// TwinCAT 3 PLC project Tc3_mxAutomationSample
// ProgramVersion: 3.1.4020.4
// libraries:
//   CmpBitmapPool, * (System)
//   Tc2_Standard, * (Beckhoff Automation GmbH)
//   Tc2_System, * (Beckhoff Automation GmbH)
//   Tc2_Utilities, * (Beckhoff Automation GmbH)
//   Tc3_Module, * (Beckhoff Automation GmbH)
//   Tc3_mxAutomationV3_0, * (Beckhoff Automation GmbH)
//   VisuDialogs, * (System)
// project tree:
//   DUTs/Diagnosis/Enum/ E_ExecMode.TcDUT, E_MoveMode.TcDUT, E_MxAStatus.TcDUT, E_MxA_Error.TcDUT, E_MxA_PCOSError.TcDUT, E_MxA_PLCError.TcDUT, E_MxA_RIError.TcDUT, E_MxA_SIError.TcDUT, E_OriType.TcDUT
//   DUTs/Diagnosis/ ST_AutoExtern.TcDUT, ST_Diag.TcDUT, ST_DiagKRC.TcDUT, ST_ErrorKRC.TcDUT, ST_FromKRC_AutoExtern.TcDUT, ST_FromKRC_P1.TcDUT, ST_GeneralKRCError.TcDUT, ST_ToKRC_AutoExtern.TcDUT, ST_ToKRC_P1.TcDUT, ST_Version.TcDUT
//   DUTs/ Robot_FW.TcDUT, Robot_Position.TcDUT
//   / GlobalTextList.TcGTLO, PlcTask.TcTTO, Visualization Manager.TcVMO (not stored), VISU_TASK.TcTTO
//   GVLs/ GVL_GUI.TcGVL, GVL_PLC.TcGVL, GVL.TcGVL, GVL_SAFETY.TcGVL, GVL_settings.TcGVL
//   POUs/ CheckBounds.TcPOU, Prg_KillHMI.TcPOU (excluded from build)
//   POUs/mxAutomation/ FB_AutoDemo.TcPOU, MAIN.TcPOU, mxA_Motion.TcPOU, Read_Axes_Velocity.TcPOU
//   POUs/Safety/ FB_SafePower.TcPOU, PRG_Safety.TcPOU
//   VISUs/ APP_Settings.TcVIS, diagnostic.TcVIS, communication.TcVIS, ImagePool.TcIPO (not stored), Motion_Axes.TcVIS, Motion_Linear.TcVIS, Motion_FBK.TcVIS, MenuMain.TcVIS, MenuTop.TcVIS, HMI_dmeo.TcVIS, MainScreen.TcVIS
//   VISUs/Text Lists/ CoorSys.TcTLO, GlobalPositions.TcTLO, ToolNumber.TcTLO
// real-time tasks:
//   TASK PlcTask: cycle T#10ms, priority 20, ADS port 350
//   TASK VISU_TASK: cycle T#50000us, priority 30, ADS port 351
// I/O:
//   DEVICE Device 3 (EtherCAT), AmsNetId 5.59.135.8.4.1
//     Box 1 (KRC4 secondary EL6695-1001) [KRC4 secondary EL6695-1001]
//       modules: Module 1 (Sync Inputs), Module 2 (Safety Data Bitf  (8 Byte)), Module 3 (Default IO)
//   DEVICE Device 1 (EtherCAT), AmsNetId 5.59.135.8.2.1
//     Term 2 (EK1200) [EK1200-5000 EtherCAT Power supply (2A E-Bus)]
//       Term 3 (EL1918) [EL1918, 8Ch. Safety Input 24V, TwinSAFE]
//         modules: Module 2 (FSLOGIC)
// variable links:
//   Device 1 (EtherCAT) <-> Device 3 (EtherCAT)/Box 1 (KRC4 secondary EL6695-1001)
//     Term 2 (EK1200)/Term 3 (EL1918)/ConnectionInputs/Message_40 TxPDO <-> Module 2 (Safety Data Bitf  (8 Byte))/Outputs Bitf/FSOE
//   Device 3 (EtherCAT) <-> Device 1 (EtherCAT)/Term 2 (EK1200)/Term 3 (EL1918)
//     Box 1 (KRC4 secondary EL6695-1001)/Module 2 (Safety Data Bitf  (8 Byte))/Inputs Bitf/FSOE <-> ConnectionOutputs/Message_40 RxPDO
//   Tc3_mxAutomationSample Instance <-> Device 1 (EtherCAT)/Term 2 (EK1200)/Term 3 (EL1918)
//     PlcTask Inputs/GVL_SAFETY.ComErr <-> StandardInputs/Standard Out Var 15
//     PlcTask Inputs/GVL_SAFETY.PowerIsOn <-> StandardInputs/Standard Out Var 42
//     PlcTask Outputs/GVL_SAFETY.Ack <-> StandardOutputs/Standard In Var 1
//     PlcTask Outputs/GVL_SAFETY.Restart <-> StandardOutputs/Standard In Var 18
//     PlcTask Outputs/GVL_SAFETY.Run <-> StandardOutputs/Standard In Var 14
//   Tc3_mxAutomationSample Instance <-> Device 3 (EtherCAT)/Box 1 (KRC4 secondary EL6695-1001)
//     PlcTask Inputs/GVL.mxIn <-> Module 3 (Default IO)/Std. In (256 Bytes)/Input DWORD 0
//     PlcTask Inputs/GVL.mxIn @bit {32..2016 step 32} <-> Module 3 (Default IO)/Std. In (256 Bytes)/Input DWORD {1..63}  (63 links)
//     PlcTask Outputs/GVL.mxOut <-> Module 3 (Default IO)/Std. Out (256 Bytes)/Output DWORD 0
//     PlcTask Outputs/GVL.mxOut @bit {32..2016 step 32} <-> Module 3 (Default IO)/Std. Out (256 Bytes)/Output DWORD {1..63}  (63 links)

CONFIGURATION Tc3_mxAutomationSample
    RESOURCE PLC ON TwinCAT3
        TASK PlcTask(INTERVAL := T#10ms, PRIORITY := 20);
        TASK VISU_TASK(INTERVAL := T#50000us, PRIORITY := 30);
        PROGRAM MAIN WITH PlcTask : MAIN;
        PROGRAM VisuElems_Visu_Prg WITH VISU_TASK : VisuElems.Visu_Prg;
    END_RESOURCE
END_CONFIGURATION

// ---- DUTs/Diagnosis/Enum/E_ExecMode.TcDUT
TYPE E_ExecMode :
(
	eEM_Submit 		:= 0, 	//direct execution, 0
	eEM_Aborting	:= 1,	//1
	eEM_Buffered	:= 2	//2
) BYTE;
END_TYPE

// ---- DUTs/Diagnosis/Enum/E_MoveMode.TcDUT
TYPE E_MoveMode :
(
	eMM_MoveAxisAbsolute := 0,
	eMM_MoveRobLinearAbsolute
);
END_TYPE

// ---- DUTs/Diagnosis/Enum/E_MxAStatus.TcDUT
TYPE E_MxAStatus :
(
	eMxA_Invalid := 0,
	eMxA_Error,
	eMxA_ProgramStopped,
	eMxA_StandBy,
	eMxA_Executing,
	eMxA_Aborting
);
END_TYPE

// ---- DUTs/Diagnosis/Enum/E_MxA_Error.TcDUT
TYPE E_MxA_Error :
(
	eMxA_OK 				:= 0, 

	eMxA_SI_InternalError,  	
	eMxA_SI_AssertFailed,		
	eMxA_SI_OvrflwStatRetQueueMain,
	eMxA_SI_OvrflwStatRetQueueTrig,
	eMxA_SI_InvCmdQueueIndex,
	eMxA_SI_InvCmdState,
	eMxA_SI_InvCmdID,
	eMxA_SI_InvMoveType,
	eMxA_SI_TrigFifoFull,
	eMxA_SI_TrigFifoEmpty,
	eMxA_SI_InvTrigFifoIndex,
	eMxA_SI_ExecOfTAfterMiss,
	eMxA_SI_ExecOfTStartMiss,
	eMxA_SI_InvAdvAct,
	eMxA_SI_AbortReq,
	eMxA_SI_TmoutHeartbeatFromPlc 	:= 16,
	eMxA_SI_InvPtpApo 				:= 30,
	eMxA_SI_InvCpApo,
	eMxA_SI_InvBaseNo,
	eMxA_SI_InvToolNo,
	eMxA_SI_InvVelo,
	eMxA_SI_InvAccel,
	eMxA_SI_InvCPtp,
	eMxA_SI_InvCDis,
	eMxA_SI_InvCVelo,
	eMxA_SI_InvCOri,
	eMxA_SI_InvOriType,
	eMxA_SI_PosDataNotInit,
	eMxA_SI_AxisPosDataNotInit,
	eMxA_SI_InvTrigDis,
	eMxA_SI_InvTrigIO,
	eMxA_SI_InvTrigPulse,
	eMxA_SI_InvCircHP,
	eMxA_SI_InvIntIO,
	eMxA_SI_InvIntPrio,
	eMxA_SI_IntNotDecl,
	eMxA_SI_InvIntAct,
	eMxA_SI_InvIONo,
	eMxA_SI_InvPulseDuration,
	eMxA_SI_InvBufferMode,
	eMxA_SI_InvToolNoForDataLoad,
	eMxA_SI_InvAnalogIONo,
	eMxA_SI_InvIpoMode,
	eMxA_SI_InvCircType,
	eMxA_SI_InvFrameData,
	eMxA_SI_InvLodaData,
	eMxA_SI_InvSoftEndRev,
	eMxA_SI_InvIntState,
	eMxA_SI_InvSysVarIndex,
	eMxA_SI_InvSysVarValue,
	eMxA_SI_SysVarNotWritable,
	eMxA_SI_InvRealValue,
	eMxA_SI_ErrorSettingOutput,
	eMxA_SI_ErrorSettingSoftEnd,
	eMxA_SI_InvTechFuncIndex,
	eMxA_SI_InvTechFuncPar,
	eMxA_SI_ParValue,

	eMxA_RI_InternalError		:= 401,	
	eMxA_RI_AssertFailed,
	eMxA_RI_InvCmdID,
	eMxA_RI_InvCmdState,
	eMxA_RI_OvrflwCmdQueue,
	eMxA_RI_IncCmdQueueIndex,
	eMxA_RI_InvCmdPreQueueIndex,
	eMxA_RI_InvWriteQueueIndex,
	eMxA_RI_StatusRetQueueSubmFull,
	eMxA_RI_InvFldbusTelLen,
	eMxA_RI_TmoutAbortReq,
	eMxA_RI_InvChkSumPlcToKrc	:= 412,
	eMxA_RI_InvMoveType,
	eMxA_RI_TmoutHeartbeatFromPlc,	
	eMxA_RI_SysVarNotInit		:= 416,
	eMxA_RI_UndflwOfNibble,
	eMxA_RI_OvrflwOfNibble,
	eMxA_RI_UndflwOfByte,
	eMxA_RI_OvrflwOfByte,
	eMxA_RI_UndflwOfInt16,
	eMxA_RI_OvrflwOfInt16,
	eMxA_RI_UndflwOfInt32,
	eMxA_RI_OvrflwOfInt32,
	eMxA_RI_UndflwOfReal,
	eMxA_RI_OvrflwOfReal,
	eMxA_RI_InvPtpApo 			:= 430,
	eMxA_RI_InvCpApo,
	eMxA_RI_InvBasNo,
	eMxA_RI_InvToolNo,
	eMxA_RI_InvVelo,
	eMxA_RI_InvAccel,
	eMxA_RI_InvCPtp,
	eMxA_RI_InvCDis,
	eMxA_RI_InvCVelo,
	eMxA_RI_InvCOri,
	eMxA_RI_InvOriType,
	eMxA_RI_PosDataNotInit,
	eMxA_RI_AxisPosDataNotInit,
	eMxA_RI_InvTrigDis,
	eMxA_RI_InvTrigIO,
	eMxA_RI_InvTrigPulse,
	eMxA_RI_InvCircHP,
	eMxA_RI_InvIntIO,
	eMxA_RI_InvIntPrio,
	eMxA_RI_IntNotDecl,
	eMxA_RI_InvIntAct,
	eMxA_RI_InvIONo,
	eMxA_RI_InvPulseDuration,
	eMxA_RI_InvBufferMode,
	eMxA_RI_InvToolNoForDataLoad,
	eMxA_RI_InvAnalogIONo,
	eMxA_RI_InvIpoMode,
	eMxA_RI_InvCircType,
	eMxA_RI_InvFrameData,
	eMxA_RI_InvLodaData,
	eMxA_RI_InvSoftEndRev,
	eMxA_RI_InvIntState,
	eMxA_RI_InvSysVarIndex,
	eMxA_RI_InvSysVarValue,
	eMxA_RI_SysVarNotWritable,
	eMxA_RI_InvRealValue,
	eMxA_RI_ErrorSettingOutput,
	eMxA_RI_ErrorSettingSoftEnd,
	eMxA_RI_InvTechFuncIndex,
	eMxA_RI_InvTechFuncPar,
	eMxA_RI_ParValue,

	eMxA_PLC_InternalError		:= 501,
	eMxA_PLC_InvBufferMode,
	eMxA_PLC_InvMxaVer,
	eMxA_PLC_InvOverride,
	eMxA_PLC_InvGrpRefIndexReached,
	eMxA_PLC_InvGrpPrefIndex,
	eMxA_PLC_InvFBOrder,
	eMxA_PLC_ConnectNotInit,
	eMxA_PLC_NoConnectToKrc,
	eMxA_PLC_TmoutHeartbeatFromKrc,
	eMxA_PLC_TmoutCmdItfBlocked,
	eMxA_PLC_InvChkSumKrcToPlc,
	eMxA_PLC_InvPosIndex,
	eMxA_PLC_PosActInv,
	eMxA_PLC_PNetError,
	eMxA_PLC_ENetIpError,
	eMxA_PLC_InvCmdSize,
	
	eMxA_PCOS_InternalError		:= 701,
	eMxA_PCOS_AssertFailed,
	eMxA_PCOS_InvCmdID,
	eMxA_PCOS_InvHeaderData,
	eMxA_PCOS_InvChkSumPlcToKrc	:= 712,
	eMxA_PCOS_InvMoveType,
	eMxA_PCOS_InvPtpApo			:= 730,
	eMxA_PCOS_InvCpApo,
	eMxA_PCOS_InvBasNo,
	eMxA_PCOS_InvToolNo,
	eMxA_PCOS_InvVelo,
	eMxA_PCOS_InvAccel,
	eMxA_PCOS_InvCPtp,
	eMxA_PCOS_InvCDis,
	eMxA_PCOS_InvCVelo,
	eMxA_PCOS_InvCOri,
	eMxA_PCOS_InvOriType,
	eMxA_PCOS_PosDataNotInit,
	eMxA_PCOS_AxisPosDataNotInit,
	eMxA_PCOS_InvTrigDis,
	eMxA_PCOS_InvTrigIO,
	eMxA_PCOS_InvTrigPulse,
	eMxA_PCOS_InvCircHP,
	eMxA_PCOS_InvIntIO,
	eMxA_PCOS_InvIntPrio,
	eMxA_PCOS_InvIntAct		:= 750,
	eMxA_PCOS_InvIONo,
	eMxA_PCOS_InvPulseDuration,
	eMxA_PCOS_InvBufferMode,
	eMxA_PCOS_InvToolNoForDataLoad,
	eMxA_PCOS_InvAnalogIONo,
	eMxA_PCOS_InvIpoMode,
	eMxA_PCOS_InvCircType,
	eMxA_PCOS_InvFrameData,
	eMxA_PCOS_InvLodaData,
	eMxA_PCOS_InvSoftEndRev,
	eMxA_PCOS_InvRealValue	:= 765,
	eMxA_PCOS_ParValue		:= 770
) DINT;
END_TYPE

// ---- DUTs/Diagnosis/Enum/E_MxA_PCOSError.TcDUT
TYPE E_MxA_PCOSError :
(
	eMxA_OK 				:= 0, 	
	eMxA_InternalError		:= 701,
	eMxA_AssertFailed,
	eMxA_InvCmdID,
	eMxA_InvHeaderData,
	eMxA_InvChkSumPlcToKrc	:= 712,
	eMxA_InvMoveType,
	eMxA_InvPtpApo			:= 730,
	eMxA_InvCpApo,
	eMxA_InvBasNo,
	eMxA_InvToolNo,
	eMxA_InvVelo,
	eMxA_InvAccel,
	eMxA_InvCPtp,
	eMxA_InvCDis,
	eMxA_InvCVelo,
	eMxA_InvCOri,
	eMxA_InvOriType,
	eMxA_PosDataNotInit,
	eMxA_AxisPosDataNotInit,
	eMxA_InvTrigDis,
	eMxA_InvTrigIO,
	eMxA_InvTrigPulse,
	eMxA_InvCircHP,
	eMxA_InvIntIO,
	eMxA_InvIntPrio,
	eMxA_InvIntAct		:= 750,
	eMxA_InvIONo,
	eMxA_InvPulseDuration,
	eMxA_InvBufferMode,
	eMxA_InvToolNoForDataLoad,
	eMxA_InvAnalogIONo,
	eMxA_InvIpoMode,
	eMxA_InvCircType,
	eMxA_InvFrameData,
	eMxA_InvLodaData,
	eMxA_InvSoftEndRev,
	eMxA_InvRealValue	:= 765,
	eMxA_ParValue		:= 770
) DINT;
END_TYPE

// ---- DUTs/Diagnosis/Enum/E_MxA_PLCError.TcDUT
TYPE E_MxA_PLCError :
(
	eMxA_OK 				:= 0, 	
	eMxA_InternalError		:= 501,
	eMxA_InvBufferMode,
	eMxA_InvMxaVer,
	eMxA_InvOverride,
	eMxA_InvGrpRefIndexReached,
	eMxA_InvGrpPrefIndex,
	eMxA_InvFBOrder,
	eMxA_ConnectNotInit,
	eMxA_NoConnectToKrc,
	eMxA_TmoutHeartbeatFromKrc,
	eMxA_TmoutCmdItfBlocked,
	eMxA_InvChkSumKrcToPlc,
	eMxA_InvPosIndex,
	eMxA_PosActInv,
	eMxA_PNetError,
	eMxA_ENetIpError,
	eMxA_InvCmdSize
) DINT;
END_TYPE

// ---- DUTs/Diagnosis/Enum/E_MxA_RIError.TcDUT
TYPE E_MxA_RIError :
(
	eMxA_OK 				:= 0, 	
	eMxA_InternalError		:= 401,	
	eMxA_AssertFailed,
	eMxA_InvCmdID,
	eMxA_InvCmdState,
	eMxA_OvrflwCmdQueue,
	eMxA_IncCmdQueueIndex,
	eMxA_InvCmdPreQueueIndex,
	eMxA_InvWriteQueueIndex,
	eMxA_StatusRetQueueSubmFull,
	eMxA_InvFldbusTelLen,
	eMxA_TmoutAbortReq,
	eMxA_InvChkSumPlcToKrc	:= 412,
	eMxA_InvMoveType,
	eMxA_TmoutHeartbeatFromPlc,	
	eMxA_SysVarNotInit		:= 416,
	eMxA_UndflwOfNibble,
	eMxA_OvrflwOfNibble,
	eMxA_UndflwOfByte,
	eMxA_OvrflwOfByte,
	eMxA_UndflwOfInt16,
	eMxA_OvrflwOfInt16,
	eMxA_UndflwOfInt32,
	eMxA_OvrflwOfInt32,
	eMxA_UndflwOfReal,
	eMxA_OvrflwOfReal,
	eMxA_InvPtpApo 			:= 430,
	eMxA_InvCpApo,
	eMxA_InvBasNo,
	eMxA_InvToolNo,
	eMxA_InvVelo,
	eMxA_InvAccel,
	eMxA_InvCPtp,
	eMxA_InvCDis,
	eMxA_InvCVelo,
	eMxA_InvCOri,
	eMxA_InvOriType,
	eMxA_PosDataNotInit,
	eMxA_AxisPosDataNotInit,
	eMxA_InvTrigDis,
	eMxA_InvTrigIO,
	eMxA_InvTrigPulse,
	eMxA_InvCircHP,
	eMxA_InvIntIO,
	eMxA_InvIntPrio,
	eMxA_IntNotDecl,
	eMxA_InvIntAct,
	eMxA_InvIONo,
	eMxA_InvPulseDuration,
	eMxA_InvBufferMode,
	eMxA_InvToolNoForDataLoad,
	eMxA_InvAnalogIONo,
	eMxA_InvIpoMode,
	eMxA_InvCircType,
	eMxA_InvFrameData,
	eMxA_InvLodaData,
	eMxA_InvSoftEndRev,
	eMxA_InvIntState,
	eMxA_InvSysVarIndex,
	eMxA_InvSysVarValue,
	eMxA_SysVarNotWritable,
	eMxA_InvRealValue,
	eMxA_ErrorSettingOutput,
	eMxA_ErrorSettingSoftEnd,
	eMxA_InvTechFuncIndex,
	eMxA_InvTechFuncPar,
	eMxA_ParValue
) DINT;
END_TYPE

// ---- DUTs/Diagnosis/Enum/E_MxA_SIError.TcDUT
TYPE E_MxA_SIError :
(
	eMxA_OK 					:= 0, 	
	eMxA_InternalError,  	
	eMxA_AssertFailed,		
	eMxA_OvrflwStatRetQueueMain,
	eMxA_OvrflwStatRetQueueTrig,
	eMxA_InvCmdQueueIndex,
	eMxA_InvCmdState,
	eMxA_InvCmdID,
	eMxA_InvMoveType,
	eMxA_TrigFifoFull,
	eMxA_TrigFifoEmpty,
	eMxA_InvTrigFifoIndex,
	eMxA_ExecOfTAfterMiss,
	eMxA_ExecOfTStartMiss,
	eMxA_InvAdvAct,
	eMxA_AbortReq,
	eMxA_TmoutHeartbeatFromPlc 	:= 16,
	eMxA_InvPtpApo 				:= 30,
	eMxA_InvCpApo,
	eMxA_InvBaseNo,
	eMxA_InvToolNo,
	eMxA_InvVelo,
	eMxA_InvAccel,
	eMxA_InvCPtp,
	eMxA_InvCDis,
	eMxA_InvCVelo,
	eMxA_InvCOri,
	eMxA_InvOriType,
	eMxA_PosDataNotInit,
	eMxA_AxisPosDataNotInit,
	eMxA_InvTrigDis,
	eMxA_InvTrigIO,
	eMxA_InvTrigPulse,
	eMxA_InvCircHP,
	eMxA_InvIntIO,
	eMxA_InvIntPrio,
	eMxA_IntNotDecl,
	eMxA_InvIntAct,
	eMxA_InvIONo,
	eMxA_InvPulseDuration,
	eMxA_InvBufferMode,
	eMxA_InvToolNoForDataLoad,
	eMxA_InvAnalogIONo,
	eMxA_InvIpoMode,
	eMxA_InvCircType,
	eMxA_InvFrameData,
	eMxA_InvLodaData,
	eMxA_InvSoftEndRev,
	eMxA_InvIntState,
	eMxA_InvSysVarIndex,
	eMxA_InvSysVarValue,
	eMxA_SysVarNotWritable,
	eMxA_InvRealValue,
	eMxA_ErrorSettingOutput,
	eMxA_ErrorSettingSoftEnd,
	eMxA_InvTechFuncIndex,
	eMxA_InvTechFuncPar,
	eMxA_ParValue
) DINT;
END_TYPE

// ---- DUTs/Diagnosis/Enum/E_OriType.TcDUT
TYPE E_OriType :
(
	eOT_Var := 0,
	eOT_Constant,
	eOT_Joint
);
END_TYPE

// ---- DUTs/Diagnosis/ST_AutoExtern.TcDUT
TYPE ST_AutoExtern :
STRUCT
	bValid				: bool;
	bRcReady			: BOOL;
	bAlarmStop			: BOOL;
	bUserSAFE			: BOOL;
	bPeriReady			: BOOL;
	bRobCal				: BOOL;
	bIoActConf			: BOOL;
	bStopMess			: BOOL;
	bIntEStop			: BOOL;
	bProAct				: BOOL;
	bApplRun			: BOOL;
	bProMove			: BOOL;
	bOnPath				: BOOL;
	bNearPosRet			: BOOL;
	bRobStopped			: BOOL;
	bT1					: BOOL;
	bT2					: BOOL;
	bAUT				: BOOL;
	bEXT				: BOOL;
END_STRUCT
END_TYPE

// ---- DUTs/Diagnosis/ST_Diag.TcDUT
TYPE ST_Diag :
STRUCT
	//KRC diag
	stDiagKRC			: ST_DiagKRC;	
	bDiagKRCError       : BOOL;
	nDiagKRCErrorID     : E_MxA_Error;
		
	//MXA error
	bMXAError           : BOOL;
	nMXAErrorID         : E_MxA_Error;
	
	//MXA status
	nMXAStatus       	: E_MxAStatus;
	bMXAStatusError     : BOOL;
	nMXAStatusErrorID   : E_MxA_Error;

	//KRC error
	stErrorKRC			: ST_ErrorKRC;
	bErrorKRCDone       : BOOL;
	bErrorKRCError      : BOOL;
	nErrorKRCErrorID    : E_MxA_Error;
END_STRUCT
END_TYPE

// ---- DUTs/Diagnosis/ST_DiagKRC.TcDUT
TYPE ST_DiagKRC :
STRUCT
	bValid         		: BOOL;
	nQueueCount         : INT;
	bPosActValid        : BOOL;
	bBrakeActive        : BOOL;
	nSubmitHeartbeat    : INT;
	nSubmitCyc_Act      : INT;
	nSubmitCyc_Min      : INT;
	nSubmitCyc_Max      : INT;
	nSubmitCyc_Avg      : INT;
	nActivePosOrderID   : DINT;
	nActiveOrderIDB     : DINT;
	nAvg_Duration       : DINT; 
	nPCOSHeartbeat 	 	: INT;   
	nPCOSCyc_Act   	 	: INT;
	nPCOSCyc_Min    	: INT;
	nPCOSCyc_Max  	  	: INT;
	nPCOSCyc_Avg    	: INT;
	nErrorID_RI         : E_MxA_RIError;
	nErrorID_SI         : E_MxA_RIError;
	nErrorID_PLC        : E_MxA_PLCError;
	nErrorID_PCOS       : E_MxA_PCOSError;
END_STRUCT
END_TYPE

// ---- DUTs/Diagnosis/ST_ErrorKRC.TcDUT
TYPE ST_ErrorKRC :
STRUCT
	bStopMessage   		: BOOL;
	nMessageCount 		: INT;
	nMessage     		: ARRAY [1..10] OF E_MxA_Error;
END_STRUCT
END_TYPE

// ---- DUTs/Diagnosis/ST_FromKRC_AutoExtern.TcDUT
TYPE ST_FromKRC_AutoExtern :
STRUCT
	bRcReady			: BOOL;	//0.0
	bAlarmStop			: BOOL;	//0.1
	bUserSAFE			: BOOL;	//0.2
	bPeriReady			: BOOL;	//0.3
	bRobCal				: BOOL;	//0.4
	bIoActConf			: BOOL;	//0.5
	bStopMess			: BOOL;	//0.6
	bPgNoFBitRefl		: BOOL;	//0.7
	
	bIntEStop			: BOOL;	//1.0
	bProAct				: BOOL;	//1.1
	bPgNoReq			: BOOL;	//1.2
	bApplRun			: BOOL;	//1.3
	bProMove			: BOOL;	//1.4
	bInHome				: BOOL;	//1.5
	bOnPath				: BOOL;	//1.6
	bNearPosRet			: BOOL;	//1.7
	
	bRobStopped			: BOOL;	//2.0
	bT1					: BOOL;	//2.1
	bT2					: BOOL;	//2.2
	bAUT				: BOOL;	//2.3
	bEXT				: BOOL;	//2.4
	bBrakeTestMonTime	: BOOL;	//2.5
	bBrakeTestReqInt	: BOOL;	//2.6
	bBrakeTestWork		: BOOL;	//2.7
	
	bBrakeTestOK		: BOOL;	//3.0
	bBrakeTestWarn		: BOOL;	//3.1
	bReserve2075		: BOOL;	//3.2
	bBrakeActive		: BOOL;	//3.3
	bKcpConnect			: BOOL;	//3.4
	bTouchUp			: BOOL;	//3.5
	bMasTestReqInt		: BOOL;	//3.6
	bMasTestSwitchOK	: BOOL;	//3.7
END_STRUCT
END_TYPE

// ---- DUTs/Diagnosis/ST_FromKRC_P1.TcDUT
{attribute 'pack_mode' := '1'}
TYPE ST_FromKRC_P1 :
STRUCT
	nStatusDw 			: DWORD;	//0
	nHeartbeatSubmit 	: BYTE;		//4		heartbeat from KRC 1..245
	nInVal_1_8			: BYTE;		//5		Actual Value of Inputs $IN[1]..$IN[8]
	nTouchUpPosNo		: INT;		//6		Position Number for TouchUp (UserTech)
	nSR_Order1_ID		: DINT;		//8		Order ID for feedback of status information
	nSR_Order2_ID		: DINT;		//12	Order ID for feedback of status information
	nSR_Order3_ID		: DINT;		//16	Order ID for feedback of status information
	nSR_Order4_ID		: DINT;		//20	Order ID for feedback of status information
	nSR_Order5_ID		: DINT;		//24	Order ID for feedback of status information
	nSR_Order6_ID		: DINT;		//28	Order ID for feedback of status information
	nSR_Order7_ID		: DINT;		//32	Order ID for feedback of status information
	nSR_Order8_ID		: DINT;		//36	Order ID for feedback of status information
	nSR_Order9_ID		: DINT;		//40	Order ID for feedback of status information
	nSR_Order10_ID		: DINT;		//44	Order ID for feedback of status information
	nSR_Order1_State	: BYTE;		//48	status feedback (in combination with nSR_Order1_ID)	
	nSR_Order2_State	: BYTE;		//49	status feedback (in combination with nSR_Order2_ID)	
	nSR_Order3_State	: BYTE;		//50	status feedback (in combination with nSR_Order3_ID)	
	nSR_Order4_State	: BYTE;		//51	status feedback (in combination with nSR_Order4_ID)	
	nSR_Order5_State	: BYTE;		//52	status feedback (in combination with nSR_Order5_ID)	
	nSR_Order6_State	: BYTE;		//53	status feedback (in combination with nSR_Order6_ID)	
	nSR_Order7_State	: BYTE;		//54	status feedback (in combination with nSR_Order7_ID)	
	nSR_Order8_State	: BYTE;		//55	status feedback (in combination with nSR_Order8_ID)	
	nSR_Order9_State	: BYTE;		//56	status feedback (in combination with nSR_Order9_ID)	
	nSR_Order10_State	: BYTE;		//57	status feedback (in combination with nSR_Order10_ID)	
	bPosActValid		: BOOL;		//58.0	Position data valid (SAK)
	nHeartbeatPCOS		: BYTE;		//59	heartbeat from PCOS 1..245
	nOverride			: BYTE;		//60	SysVar $OV_PRO
	fPosActX			: REAL;		//61	SysVar $POS_ACT.X
	fPosActY			: REAL;		//65	SysVar $POS_ACT.Y
	fPosActZ			: REAL;		//69	SysVar $POS_ACT.Z
	fPosActA			: REAL;		//73	SysVar $POS_ACT.A
	fPosActB			: REAL;		//77	SysVar $POS_ACT.B
	fPosActC			: REAL;		//81	SysVar $POS_ACT.C
	nPosActStatus		: DINT;		//85	SysVar $POS_ACT.S
	nPosActTurns		: BYTE;		//89	SysVar $POS_ACT.T
	nToolAct			: SINT;		//90	SysVar $ACT_TOOL_C
	nBaseAct			: SINT;		//91	SysVar $ACT_BASE_C
	nIpoMode			: BYTE;		//92	SysVar $IPO_MODE_C
	fAxisAct_A1			: REAL;		//93	SysVar $AXIS_ACT.A1
	fAxisAct_A2			: REAL;		//97	SysVar $AXIS_ACT.A2
	fAxisAct_A3			: REAL;		//101	SysVar $AXIS_ACT.A3
	fAxisAct_A4			: REAL;		//105	SysVar $AXIS_ACT.A4
	fAxisAct_A5			: REAL;		//109	SysVar $AXIS_ACT.A5
	fAxisAct_A6			: REAL;		//113	SysVar $AXIS_ACT.A6
	fAxisAct_A7			: REAL;		//117	SysVar $AXIS_ACT.A7
	fAxisAct_A8			: REAL;		//121	SysVar $AXIS_ACT.A8
	fAxisAct_A9			: REAL;		//125	SysVar $AXIS_ACT.A9
	fAxisAct_A10		: REAL;		//129	SysVar $AXIS_ACT.A10
	fAxisAct_A11		: REAL;		//133	SysVar $AXIS_ACT.A11
	fAxisAct_A12		: REAL;		//137	SysVar $AXIS_ACT.A12
	fVelAct				: REAL;		//141	SysVar $VEL_ACT
	nVelAxis_A1			: SINT;		//145	SysVar $VEL_AXIS_ACT[1]
	nVelAxis_A2			: SINT;		//146	SysVar $VEL_AXIS_ACT[2]
	nVelAxis_A3			: SINT;		//147	SysVar $VEL_AXIS_ACT[3]
	nVelAxis_A4			: SINT;		//148	SysVar $VEL_AXIS_ACT[4]
	nVelAxis_A5			: SINT;		//149	SysVar $VEL_AXIS_ACT[5]
	nVelAxis_A6			: SINT;		//150	SysVar $VEL_AXIS_ACT[6]
	nVelAxis_A7			: SINT;		//151	SysVar $VEL_AXIS_ACT[7]
	nVelAxis_A8			: SINT;		//152	SysVar $VEL_AXIS_ACT[8]
	nVelAxis_A9			: SINT;		//153	SysVar $VEL_AXIS_ACT[9]
	nVelAxis_A10		: SINT;		//154	SysVar $VEL_AXIS_ACT[10]
	nVelAxis_A11		: SINT;		//155	SysVar $VEL_AXIS_ACT[11]
	nVelAxis_A12		: SINT;		//156	SysVar $VEL_AXIS_ACT[12]
	nGroupState			: BYTE;		//157	see state diagram
	nErrorId			: INT;		//158	error id from main loop or interrupt
	nErrorSubId			: INT;		//160	error id from submit interpreter
	nActivePosOrderId	: DINT;		//162	order id of active move cmd
	nActiveOrderIdB		: DINT;		//166	active order id in preparation
	nQueueCount			: BYTE;		//170	current amount of functions in buffer
	nIR_Status_1_2		: BYTE;		//171	status of interrupt 1 and 2
	nIR_Status_3_4		: BYTE;		//172	status of interrupt 3 and 4
	nIR_Status_5_6		: BYTE;		//173	status of interrupt 5 and 6
	nIR_Status_7_8		: BYTE;		//174	status of interrupt 7 and 8
	nErrorIdPCOS		: BYTE;		//175	error id of ProConOS
	nFreeForMove		: BYTE;		//176	reserved for ProConOS
	nTransmissionNoNet	: BYTE;		//177	acknowledge of transmission number
	nOrderIdRet			: DINT;		//178	acknowledge take data of cmd
	nCmdIdRet			: DINT;		//182	acknowledge take data of cmd
	nCmdDataRetCS		: DINT;		//186	checksum data feedback
	nReserved190		: DINT;		//190	reserved
	fCmdDataRet1		: REAL;		//194	command dependent	
	fCmdDataRet2		: REAL;		//198	command dependent	
	fCmdDataRet3		: REAL;		//202	command dependent	
	fCmdDataRet4		: REAL;		//206	command dependent	
	fCmdDataRet5		: REAL;		//210	command dependent	
	fCmdDataRet6		: REAL;		//214	command dependent	
	fCmdDataRet7		: REAL;		//218	command dependent	
	fCmdDataRet8		: REAL;		//222	command dependent	
	fCmdDataRet9		: REAL;		//226	command dependent	
	fCmdDataRet10		: REAL;		//230	command dependent	
	fCmdDataRet11		: REAL;		//234	command dependent	
	fCmdDataRet12		: REAL;		//238	command dependent
	nReserve242			: DINT;		//242	reserved	
	nReserve246			: ARRAY [1..10] OF BYTE; //246..255
END_STRUCT
END_TYPE

// ---- DUTs/Diagnosis/ST_GeneralKRCError.TcDUT
TYPE ST_GeneralKRCError :
STRUCT
	nErrorId 			: DINT;
	bNoHeartbeatKrc 	: BOOL;
	bNoHeartbeatPCOS 	: BOOL;
	bNotOnline 			: BOOL;
	bNotInitialized 	: BOOL;
	bNoOpModeExt 		: BOOL;
	bNoMoveEnable		: BOOL;
	bUserSafeNotOK		: BOOL;
	bKrcErrorActive 	: BOOL;
	bDrivesNotReady		: BOOL; 
	bNoProgActive		: BOOL;
END_STRUCT
END_TYPE

// ---- DUTs/Diagnosis/ST_ToKRC_AutoExtern.TcDUT
TYPE ST_ToKRC_AutoExtern :
STRUCT
	bPgNo_FBit			: BOOL;	//0.0
	bPgNo_Bit1			: BOOL;	//0.1
	bPgNo_Bit2			: BOOL;	//0.2
	bPgNo_Bit3			: BOOL;	//0.3
	bPgNo_Bit4			: BOOL;	//0.4
	bPgNo_Bit5			: BOOL;	//0.5
	bPgNo_Bit6			: BOOL;	//0.6
	bPgNo_Bit7			: BOOL;	//0.7
	
	bPgNo_Parity		: BOOL;	//1.0
	bPgNo_Valid			: BOOL;	//1.1
	bExtStart			: BOOL;	//1.2
	bMoveEnable			: BOOL;	//1.3
	bConfMess			: BOOL;	//1.4
	bDrivesOff			: BOOL;	//1.5
	bDrivesOn			: BOOL;	//1.6
	bMasteringTestReqExt: BOOL;	//1.7
	
	bBrakeTestReqExt	: BOOL;	//2.0
	bReserve_2_1_3_7	: ARRAY[1..15] OF BOOL; //2.1 - 3.7
	
	bReset				: BOOL;	//4.0	choose cell program with rising edge
	bBrake				: BOOL;	//4.1	brake command (KRC interrupt)
	bBrakeF				: BOOL;	//4.2	brakeF command (KRC interrupt)
	bReleaseBrake		: BOOL;	//4.3	release brake after brake command
	bShowTrace			: BOOL;	//4.4	show diag messages in message window
	bMessageReset		: BOOL;	//4.5	message aknowledge of error messages of mxAutomation package
	bReserve_4_6		: BOOL;	//4.6
	bWriteOut_1to8		: BOOL;	//4.7	write request for outputs 1 to 8
	
	bOutVal1			: BOOL;	//5.0	setvalue for $OUT[1]
	bOutVal2			: BOOL;	//5.1	setvalue for $OUT[2]
	bOutVal3			: BOOL;	//5.2	setvalue for $OUT[3]
	bOutVal4			: BOOL;	//5.3	setvalue for $OUT[4]
	bOutVal5			: BOOL;	//5.4	setvalue for $OUT[5]
	bOutVal6			: BOOL;	//5.5	setvalue for $OUT[6]
	bOutVal7			: BOOL;	//5.6	setvalue for $OUT[7]
	bOutVal8			: BOOL;	//5.7	setvalue for $OUT[8]
	
	bReserve_6_0_7_7	: ARRAY[1..16] OF BOOL; //6.0 - 7.7
END_STRUCT
END_TYPE

// ---- DUTs/Diagnosis/ST_ToKRC_P1.TcDUT
{attribute 'pack_mode' := '1'}
TYPE ST_ToKRC_P1 :
STRUCT
	nControlLw			: LWORD;	//0
	nHeartbeat			: BYTE;		//8		heartbeat KRC and ProConOS, 1..254
	nOverride			: BYTE;		//9		override of extern
	nPlcVersionMajor	: BYTE;		//10	major PLC version
	nPlcVersionMinor	: BYTE;		//11	minor PLC version
	nSR_Order1_IdRet	: DINT;		//12	order id for acknowledge of status feedback
	nSR_Order2_IdRet	: DINT;		//16	order id for acknowledge of status feedback
	nSR_Order3_IdRet	: DINT;		//20	order id for acknowledge of status feedback
	nSR_Order4_IdRet	: DINT;		//24	order id for acknowledge of status feedback
	nSR_Order5_IdRet	: DINT;		//28	order id for acknowledge of status feedback
	nSR_Order6_IdRet	: DINT;		//32	order id for acknowledge of status feedback
	nSR_Order7_IdRet	: DINT;		//36	order id for acknowledge of status feedback
	nSR_Order8_IdRet	: DINT;		//40	order id for acknowledge of status feedback
	nSR_Order9_IdRet	: DINT;		//44	order id for acknowledge of status feedback
	nSR_Order10_IdRet	: DINT;		//48	order id for acknowledge of status feedback
	nSR_Order1_State	: BYTE;		//52	order id for acknowledge of status feedback
	nSR_Order2_State	: BYTE;		//53	order id for acknowledge of status feedback
	nSR_Order3_State	: BYTE;		//54	order id for acknowledge of status feedback
	nSR_Order4_State	: BYTE;		//55	order id for acknowledge of status feedback
	nSR_Order5_State	: BYTE;		//56	order id for acknowledge of status feedback
	nSR_Order6_State	: BYTE;		//57	order id for acknowledge of status feedback
	nSR_Order7_State	: BYTE;		//58	order id for acknowledge of status feedback
	nSR_Order8_State	: BYTE;		//59	order id for acknowledge of status feedback
	nSR_Order9_State	: BYTE;		//60	order id for acknowledge of status feedback
	nSR_Order10_State	: BYTE;		//61	order id for acknowledge of status feedback
	nTransmissionNO1	: BYTE;		//62	1..254: transmission number, 0: no active transmission
	nTransmissionType	: BYTE;		//63	1: Part 1/1, 2: Part 1/2, 3: Part 2/2, 4: Part 1/3, 5: Part 2/3, 6: Part 3/3
	nOrderId			: DINT;		//64	unique order id, incr. with rising edge on bExecute on FB, 1..2^31-1
	nCmdId				: BYTE;		//68	command id
	eExecMode			: E_ExecMode;//69	Enum Byte: 0: Submit (direct execution in submit), 1: aborting, 2: buffered
	nCheckSum			: DWORD;	//70	XOR checksum of command data
	nBoolValues1		: WORD;		//74	bool parameter values 1-15, 16-30, 31-45
	nCmdParInt1			: DINT;		//76	integer parameter 1, 16, 31
	nCmdParInt2			: DINT;		//80	integer parameter 2, 17, 32
	nCmdParInt3			: DINT;		//84	integer parameter 3, 18, 33
	nCmdParInt4			: DINT;		//88	integer parameter 4, 19, 34
	nCmdParInt5			: DINT;		//92	integer parameter 5, 20, 35
	nCmdParInt6			: DINT;		//96	integer parameter 6, 21, 36
	nCmdParInt7			: DINT;		//100	integer parameter 7, 22, 37
	nCmdParInt8			: DINT;		//104	integer parameter 8, 23, 38
	nCmdParInt9			: DINT;		//108	integer parameter 9, 24, 39
	nCmdParInt10		: DINT;		//112	integer parameter 10, 25, 40
	nCmdParInt11		: DINT;		//116	integer parameter 11, 26, 41
	nCmdParInt12		: DINT;		//120	integer parameter 12, 27, 42
	nCmdParInt13		: DINT;		//124	integer parameter 13, 28, 43
	nCmdParInt14		: DINT;		//128	integer parameter 14, 29, 44
	nCmdParInt15		: DINT;		//132	integer parameter 15, 30, 45
	fCmdParReal1		: REAL;		//136	real parameter 1, 16, 31
	fCmdParReal2		: REAL;		//140	real parameter 2, 17, 32
	fCmdParReal3		: REAL;		//144	real parameter 3, 18, 33
	fCmdParReal4		: REAL;		//148	real parameter 4, 19, 34
	fCmdParReal5		: REAL;		//152	real parameter 5, 20, 35
	fCmdParReal6		: REAL;		//156	real parameter 6, 21, 36
	fCmdParReal7		: REAL;		//160	real parameter 7, 22, 37
	fCmdParReal8		: REAL;		//164	real parameter 8, 23, 38
	fCmdParReal9		: REAL;		//168	real parameter 9, 24, 39
	fCmdParReal10		: REAL;		//172	real parameter 10, 25, 40
	fCmdParReal11		: REAL;		//176	real parameter 11, 26, 41
	fCmdParReal12		: REAL;		//180	real parameter 12, 27, 42
	fCmdParReal13		: REAL;		//184	real parameter 13, 28, 43
	fCmdParReal14		: REAL;		//188	real parameter 14, 29, 44
	fCmdParReal15		: REAL;		//192	real parameter 15, 30, 45
	nTransmissionNO2	: BYTE;		//196	transmission number for consistency check, need to match with nTransmissionNO1
	nReserved197		: ARRAY [1..59] OF BYTE;	
END_STRUCT
END_TYPE

// ---- DUTs/Diagnosis/ST_Version.TcDUT
TYPE ST_Version :
STRUCT
	nMajor    		: DINT;
	nMinor    		: DINT;
	nBuild 			: DINT;
	nRevision 		: DINT;
	sVersion		: STRING;
END_STRUCT
END_TYPE

// ---- DUTs/Robot_FW.TcDUT
TYPE Robot_FW :
	
STRUCT
	FW_Version :DINT;
	FW_Major:DINT;
	FW_Minor:DINT;
	
END_STRUCT


END_TYPE

// ---- DUTs/Robot_Position.TcDUT
TYPE Robot_Position :
	

STRUCT
	
p1:REAL;
p2:REAL;
p3:REAL;
p4:REAL;
p5:REAL;
p6:REAL;

END_STRUCT


END_TYPE

// ---- GVLs/GVL_GUI.TcGVL
{attribute 'qualified_only'}
VAR_GLOBAL
	
	LinearTargetCommand :STRING;
	GlobalPositionString :STRING;

	
END_VAR

// ---- GVLs/GVL_PLC.TcGVL
{attribute 'qualified_only'}
VAR_GLOBAL
	
	Int_windowsCounter: ULINT;
	Str_windowsCounter: STRING;
	
	
	ReadWindowsTime : fb_localsystemTime;
	String_WindowsTime: STRING;
	Time_SystemTime : TIMESTRUCT;
	
END_VAR

// ---- GVLs/GVL.TcGVL
{attribute 'qualified_only'}
VAR_GLOBAL
	
//=====================================
// mxAutomation
//=====================================	

	mxIn					AT%I* 	: ARRAY[0..63] OF DWORD;
	mxOut 					AT%Q* 	: ARRAY[0..63] OF DWORD;
	
	nAxisIndex						: INT := 1;  // Robot number one, may be any unique number between 1..5
	nOverrideGlobal					: INT;
	
	stCoordSys						: COORDSYS;
	stApprox						: APO;
	
	HMI_ActualCartPos				: E6POS;
	HMI_ActualAxisPosition			: E6AXIS;
	
	HMI_AutoStart					: BOOL;
	HMI_MessageReset				: BOOL;
	
	HMI_AutoEXT						: BOOL;
	HMI_DrivesNotReady				: BOOL;
	
	HMI_Error_ProConOS				: BOOL;
	HMI_Error_SINT					: BOOL;
	HMI_Error_General				: BOOL;
	HMI_Error_General_ID			: DINT;
	
	HMI_WriteLoadData				: BOOL;
	HMI_LOAD						: INT;
	HMI_TOOL						: INT;
	HMI_BASE						: INT;
	
	HMI_TouchUpStoreNow				: BOOL;
	HMI_TouchUpIndex				: INT;
	
	in_MOVE_ENABLE					: BOOL;
	in_CONF_MESS					: BOOL;
	in_DRIVES_ON					: BOOL;
	in_DRIVES_OFF					: BOOL;
	in_EXT_START					: BOOL;
	in_ENABLE_T1					: BOOL;
	in_ENABLE_T2					: BOOL;
	in_ENABLE_AUT					: BOOL;
	in_ENABLE_EXT					: BOOL;
	
	out_ALARM_STOP					: BOOL;
	out_USER_SAFE					: BOOL;
	
	
END_VAR 
VAR_GLOBAL RETAIN
	aPosArray	 					: POSITION_ARRAY;
	LinearArray 					: POSITION_ARRAY;
	kuka_fw 						: Robot_FW;
END_VAR

// ---- GVLs/GVL_SAFETY.TcGVL
{attribute 'qualified_only'}
VAR_GLOBAL
	ComErr, EMO_Diag,PowerIsOn AT%I*:BOOL;
	Ack,Run,Restart AT%Q*:BOOL;
END_VAR

// ---- GVLs/GVL_settings.TcGVL
{attribute 'qualified_only'}
VAR_GLOBAL
	

App_Velocity : REAL;
App_Acceleration : REAL;
App_CoordSys : COORDSYS;
App_GroupIndex :INT:=1;
App_BufferMode :INT :=2;
App_APO :APO ;
App_ToolNumber :INT;


//app_coordsys.BASE:=1;
//app_coordsys.TOOL:=1;
//app_coordsys.IPO_Mode:=0;


END_VAR

// ---- POUs/mxAutomation/MAIN.TcPOU
PROGRAM MAIN
VAR
	
	fbKRC_ReadAxisGroup			: KRC_ReadAxisGroup;
	fbKRC_WriteAxisGroup		: KRC_WriteAxisGroup;
	fbKRC_Error					: KRC_Error;
	fbKRC_Diag					: KRC_Diag;
	fbKRC_AutomaticExternal		: KRC_AutomaticExternal;
	fbKRC_Initialize			: KRC_Initialize;
	fbKRC_AutoStart				: KRC_AutoStart;
	fbKRC_SetOverride			: KRC_SetOverride;
	Read_Axes_SW_Limts          : krc_readsoftend;
	Write_Program_Abort			: krc_abort;
		 
	Move_Axes 					: MC_MoveAxisAbsolute;
	Move_Linear 				: MC_MoveLinearAbsolute;
	
	bInitError					: BOOL;
	nInitErrorID				: DINT;
	bInitDone					: BOOL;
	bAutoExternReset			: BOOL;
	bAutostartDone				: BOOL;
	bAutostartResetValid		: BOOL;
	bAutostartDispActive		: BOOL;
	
	LinearTargetPOS				:E6POS;
	LinearTargetCOORD			:COORDSYS;
	inearTargetAPO				:APO;
	
	ReadKRCError 				:KRC_ReadKRCError;
	NOT_INT_E_STOP				:BOOL;
	

END_VAR

fbKRC_ReadAxisGroup(KRC4_Input := ADR(GVL.mxIn),AxisGroupIdx := GVL.nAxisIndex);

A_StartUp();
A_Diagnosis();

mxA_Motion();

move_Axes(
	axisgroupidx := gvl_settings.App_GroupIndex,
	execute := ,
	axisposition:=,
	velocity:= gvl_settings.App_Velocity ,
	acceleration := gvl_settings.App_Acceleration,
	approximate :=gvl_settings.App_APO ,
	queuemode := gvl_settings.App_BufferMode );
	
	
//gvl_settings.App_CoordSys.BASE:=1;
//gvl_settings.app_coordsys.TOOL:=1;
//gvl_settings.app_coordsys.IPO_Mode:=0;

move_Linear(
		axisgroupidx := gvl_settings.App_GroupIndex ,
		execute := ,
		position := LinearTargetPOS ,
		velocity := gvl_settings.App_Velocity ,
		acceleration :=gvl_Settings.App_Acceleration ,
		CoordinateSystem := ,///gvl_settings.App_CoordSys,
		oritype :=0 ,
		approximate:= ,//gvl_settings.App_APO,
		queuemode :=2  ,
		errorid => );

		
Read_Axes_Velocity();	


ReadKRCError(
	AxisGroupIdx:= gvl_settings.App_GroupIndex , 
	ExecuteCmd:= , 
	Offset:= , 
	Done=> , 
	Error=> , 
	ErrorID=> , 
	STOPMESS=> , 
	MessageCount=> , 
	Message1=> , 
	Message2=> , 
	Message3=> , 
	Message4=> , 
	Message5=> , 
	Message6=> , 
	Message7=> , 
	Message8=> , 
	Message9=> , 
	Message10=> );
	
fbKRC_WriteAxisGroup(AxisGroupIdx := GVL.nAxisIndex, KRC4_Output:= ADR(GVL.mxOut)); 


//--read windows counter and convert to string---
GVL_PLC.Int_windowsCounter := f_getsystemtime();
GVL_PLC.Str_windowsCounter := ULINT_TO_STRING(ABS(GVL_PLC.Int_windowsCounter));


//--read windows Date and time---
GVL_PLC.ReadWindowsTime(
	sNetID:= , 
	bEnable:=TRUE , 
	dwCycle:= 1, 
	dwOpt:= , 
	tTimeout:= , 
	bValid=> , 
	systemTime=>gvl_plc.Time_SystemTime,
	tzID=> );
	

gvl_plc.String_WindowsTime := systemtime_to_string(gvl_plc.Time_SystemTime);

ACTION A_Diagnosis:
fbKRC_Error(
	AxisGroupIdx:= GVL.nAxisIndex, 
	MessageReset:=  ,//GVL.HMI_MessageReset, 
	Error=> ,//GVL.HMI_Error_General , 
	ErrorID=> ,//GVL.HMI_Error_General_ID, 
	NoHeartbeatKRC=> , 
	NoHeartbeatPCOS=> , 
	NotOnline=> , 
	NotInitialized=> , 
	NoOpModeExt=> , 
	NoMoveEnable=> , 
	UserSafeNotOK=> , 
	KrcErrorActive=> , 
	DrivesNotReady=> , 
	NoProgActive=> );	

GVL.HMI_Error_SINT := NOT  fbKRC_Error.NoHeartbeatKRC;
GVL.HMI_Error_ProConOS := NOT fbKRC_Error.NoHeartbeatPCOS;
GVL.HMI_DrivesNotReady := NOT fbKRC_Error.DrivesNotReady;



	
fbKRC_Diag(
	AxisGroupIdx:= GVL.nAxisIndex, 
	ShowTrace:= FALSE, 
	MaxSubmitCycle:= , 
	Valid=> , 
	QueueCount=> , 
	PosActValid=> , 
	BrakeActive=> , 
	SubmitHeartbeat=> , 
	SubmitCyc_Act=> , 
	SubmitCyc_Min=> , 
	SubmitCyc_Max=> , 
	SubmitCyc_Avg=> , 
	ActivePosOrderID=> , 
	ActiveOrderIDB=> , 
	Avg_Duration=> , 
	ProconosHeartbeat=> , 
	ProconosCyc_Act=> , 
	ProconosCyc_Min=> , 
	ProconosCyc_Max=> , 
	ProconosCyc_Avg=> , 
	ErrorID_RI=> , 
	ErrorID_SI=> , 
	ErrorID_PLC=> , 
	ErrorID_PCOS=> , 
	Error=> , 
	ErrorID=> );	
	
	
	read_axes_sw_limts(
		axisgroupidx :=gvl_settings.App_GroupIndex ,
		executecmd:= ,
		done :=,
		a1_min := ,
		a1_max := ,
		a2_min := ,
		a2_max := ,
		a3_min := ,
		a3_max := ,
		a4_min := ,
		a4_max := ,
		a5_min := ,
		a5_max := ,
		a6_min := ,
		a6_max := ,
		error := ,
		errorID:=);
END_ACTION

ACTION A_StartUp:
fbKRC_Initialize(
	AxisGroupIdx:= gvl.nAxisIndex, 
	Done=> bInitDone , 
	Error=> bInitError, 
	ErrorID=>  nInitErrorID, 
	KRC_Serial=>, 
	KRC_Major=>, 
	KRC_Minor=> , 
	KRC_Revision=>, 
	PLC_Major=> , 
	PLC_Minor=>, 
	PLC_Revision=>);
	
fbKRC_AutomaticExternal(
	AxisGroupIdx:= GVL.nAxisIndex, 
	MOVE_ENABLE:=,//GVL.in_MOVE_ENABLE,//true 
	CONF_MESS:=GVL.in_CONF_MESS ,//GVL.in_CONF_MESS, 
	DRIVES_ON:= ,//GVL.in_DRIVES_ON, 
	DRIVES_OFF:= ,//=GVL.in_DRIVES_OFF ,//TRUE , 
	EXT_START:=GVL.in_EXT_START , //GVL.in_EXT_START, 
	RESET:= ,//bAutoExternReset, 
	ENABLE_T1:= ,//GVL.in_ENABLE_T1 ,//TRUE, 
	ENABLE_T2:= ,//GVL.in_ENABLE_T2 ,//TRUE, 
	ENABLE_AUT:= ,// GVL.in_ENABLE_AUT,//,TRUE, 
	ENABLE_EXT:=  ,//GVL.in_ENABLE_EXT,//TRUE, 
	Valid=> , 
	RC_RDY1=> , 
	ALARM_STOP=>GVL.out_ALARM_STOP , 
	USER_SAFE=> GVL.out_USER_SAFE, 
	PERI_RDY=> , 
	ROB_CAL=> , 
	IO_ACTCONF=> , 
	STOPMESS=> , 
	INT_E_STOP=> , 
	PRO_ACT=> , 
	APPL_RUN=> , 
	PRO_MOVE=> , 
	ON_PATH=> , 
	NEAR_POSRET=> , 
	ROB_STOPPED=> , 
	T1=> , 
	T2=> , 
	AUT=> , 
	EXT=>  );
//GVL.HMI_AutoEXT);	
	
NOT_INT_E_STOP := NOT(MAIN.fbKRC_AutomaticExternal.INT_E_STOP);	

fbKRC_AutoStart(
	AxisGroupIdx:= GVL.nAxisIndex , 
	ExecuteReset:=  ,//GVL.HMI_AutoStart, 
	Busy=> , 
	Done=> bAutostartDone, 
	DispActive=> bAutostartDispActive, 
	ResetValid=> bAutostartResetValid , 
	Error=> , 
	ErrorID=> );
	
fbKRC_SetOverride(
	AxisGroupIdx:=GVL.nAxisIndex , 
	Override:= GVL.nOverrideGlobal , 
	Valid=> , 
	ActualOverride=> , 
	Error=> , 
	ErrorID=> );	
	
write_program_abort(
		axisgroupidx :=gvl_settings.App_GroupIndex,
		executecmd := ,
		);
END_ACTION

END_PROGRAM

// ---- POUs/mxAutomation/mxA_Motion.TcPOU
PROGRAM mxA_Motion
VAR
	fbKRC_ReadActualPosition		: KRC_ReadActualPosition;
	fbKRC_ReadActualAxisPosition	: KRC_ReadActualAxisPosition;
	fbKRC_ReadActualVelocity		: KRC_ReadActualVelocity;
	
	fbKRC_TouchUP					: KRC_TouchUP;
	fbKRC_ReadTouchUPState			: KRC_ReadTouchUPState;
	fbKRC_Jog						: KRC_Jog;
	fbMC_MoveLinearAbsolute			: MC_MoveLinearAbsolute;
	fbMC_MoveDirectAbsolute			: MC_MoveDirectAbsolute;
	
	fbKRC_WriteLoadData				: KRC_WriteLoadData;
	
	fbMxa_ValuesToCOORDSYS			: mxa_ValuesToCOORDSYS;
	fbMxa_ValuesToAPO				: mxa_ValuesToAPO;
	
	nMove_PositonMode_Pos			: INT;
	bMoveLinar_PositonMode			: BOOL;
	bMovePTP_PositonMode			: BOOL;
	
	nJogMoveType					: INT := 0;
	
	bJogA1_P						: BOOL;
	bJogA1_M						: BOOL;
	bJogA2_P						: BOOL;
	bJogA2_M						: BOOL;
	bJogA3_P						: BOOL;
	bJogA3_M						: BOOL;
	bJogA4_P						: BOOL;
	bJogA4_M						: BOOL;
	bJogA5_P						: BOOL;
	bJogA5_M						: BOOL;
	bJogA6_P						: BOOL;
	bJogA6_M						: BOOL;
	
	nState							: UDINT;
	bExecAutoDemo					: BOOL;
	fbAutoDemo						: FB_AutoDemo;
END_VAR

mxA_TouchUp();
mxA_Data();

CASE nState OF
0:	
	mxA_Tool_Base();
	mxa_Jog();
	mxA_PositionMode();

	mxA_LoadData();
		 

	
	 IF bExecAutoDemo 
		AND NOT fbKRC_Jog.Busy 
		AND NOT fbMC_MoveDirectAbsolute.Busy 
		AND NOT fbMC_MoveLinearAbsolute.Busy
		AND NOT fbKRC_WriteLoadData.Busy THEN
		 nState := 10;
	 END_IF
 10:
 	fbAutoDemo(bExecute := bExecAutoDemo);
	
	IF NOT bExecAutoDemo AND NOT fbAutoDemo.bBusy THEN
		nState := 0;
	END_IF
 END_CASE

ACTION mxA_Data:

fbKRC_ReadActualPosition(
	AxisGroupIdx:= GVL.nAxisIndex , 
	Valid=> , 
	Position=> GVL.HMI_ActualCartPos, 
	X=> , 
	Y=> , 
	Z=> , 
	A=> , 
	B=> , 
	C=> , 
	Status=> , 
	Turn=> , 
	Tool=> , 
	Base=> , 
	IPOMode=> );
	
fbKRC_ReadActualAxisPosition(
	AxisGroupIdx:= GVL.nAxisIndex , 
	Valid=> , 
	AxisPosition=> GVL.HMI_ActualAxisPosition , 
	A1=> , 
	A2=> , 
	A3=> , 
	A4=> , 
	A5=> , 
	A6=> , 
	E1=> , 
	E2=> , 
	E3=> , 
	E4=> , 
	E5=> , 
	E6=> );	
	
fbKRC_ReadActualVelocity(AxisGroupIdx:= GVL.nAxisIndex , Valid=> , Value=> );
END_ACTION

ACTION mxA_Jog:
fbKRC_Jog(
	AxisGroupIdx:= GVL.nAxisIndex , 
	MoveType:= nJogMoveType, 
	Velocity:= 50, 
	Acceleration:= 50, 
	CoordinateSystem:= GVL.stCoordSys, 
	Increment:= 0.0, 
	A1_X_P:= bJogA1_P, 
	A1_X_M:= bJogA1_M, 
	A2_Y_P:= bJogA2_P, 
	A2_Y_M:= bJogA2_M, 
	A3_Z_P:= bJogA3_P, 
	A3_Z_M:= bJogA3_M, 
	A4_A_P:= bJogA4_P, 
	A4_A_M:= bJogA4_M, 
	A5_B_P:= bJogA5_P, 
	A5_B_M:= bJogA5_M, 
	A6_C_P:= bJogA6_P, 
	A6_C_M:= bJogA6_M, 
	E1_P:= , 
	E1_M:= , 
	E2_P:= , 
	E2_M:= , 
	E3_P:= , 
	E3_M:= , 
	E4_P:= , 
	E4_M:= , 
	E5_P:= , 
	E5_M:= , 
	E6_P:= , 
	E6_M:= , 
	Busy=> , 
	Active=> , 
	Done=> , 
	Aborted=> , 
	Error=> , 
	ErrorID=> );
END_ACTION

ACTION mxA_LoadData:
fbKRC_WriteLoadData(
	AxisGroupIdx:= gvl.nAxisIndex , 
	ExecuteCmd:= GVL.HMI_WriteLoadData, 
	Tool:= GVL.HMI_TOOL, 
	M:= GVL.HMI_LOAD, 
	X:= , 
	Y:= , 
	Z:= , 
	A:= , 
	B:= , 
	C:= , 
	JX:= , 
	JY:= , 
	JZ:= , 
	BufferMode:= eEM_Aborting, 
	Busy=> , 
	Done=> , 
	Aborted=> , 
	Error=> , 
	ErrorID=> );
END_ACTION

ACTION mxA_PositionMode:
fbMxa_ValuesToAPO(
	PTP_MODE:= 0, 
	CP_MODE:= 0, 
	CPTP:= , 
	CDIS:= , 
	CORI:= , 
	CVEL:= , 
	APO=> GVL.stApprox);
	
//fbMC_MoveDirectAbsolute(
//	AxisGroupIdx:= GVL.nAxisIndex, 
//	Execute:= mxA_Motion.bMovePTP_PositonMode, 
//	Position:= GVL.aPosArray[nMove_PositonMode_Pos].E6POS, 
//	Velocity:= 50, 
//	Acceleration:= 50, 
//	CoordinateSystem:= GVL.aPosArray[nMove_PositonMode_Pos].COORDSYS, 
//	Approximate:= GVL.stApprox , 
//	QueueMode:= eEM_Aborting, 
//	ComAcpt=> , 
//	ComBusy=> , 
//	Busy=> , 
//	Active=> , 
//	Done=> , 
//	CommandAborted=> , 
//	Error=> , 
//	ErrorID=> );	
	
//fbMC_MoveLinearAbsolute(
//	AxisGroupIdx:= GVL.nAxisIndex, 
//	Execute:= mxA_Motion.bMoveLinar_PositonMode , 
//	Position:= GVL.aPosArray[nMove_PositonMode_Pos].E6POS, 
//	Velocity:= 1,
//	Acceleration:= 2.3, 
//	CoordinateSystem:= GVL.stCoordSys , 
//	OriType:= 0, 
//	Approximate:= GVL.stApprox , 
//	QueueMode:= eEM_Aborting, 
//	ComAcpt=> , 
//	ComBusy=> , 
//	Busy=> , 
//	Active=> , 
//	Done=> , 
//	CommandAborted=> , 
//	Error=> , 
//	ErrorID=> );
END_ACTION

ACTION mxA_Tool_Base:
fbMxa_ValuesToCOORDSYS(
	Tool:= GVL.HMI_TOOL,
	Base:= GVL.HMI_BASE, 
	IPO_Mode:= 0,
	COORDSYS=> GVL.stCoordSys);
END_ACTION

ACTION mxA_TouchUp:

fbKRC_ReadTouchUPState(
	AxisGroupIdx:= gvl.nAxisIndex, 
	Valid=> , 
	TouchUP=> , 
	Index=> , 
	Error=> , 
	ErrorID=> );	

IF fbKRC_ReadTouchUPState.TouchUP THEN
	fbKRC_TouchUP.Index := fbKRC_ReadTouchUPState.Index;
ELSIF GVL.HMI_TouchUpStoreNow THEN
	fbKRC_TouchUP.Index := GVL.HMI_TouchUpIndex;
END_IF	
	
fbKRC_TouchUP(
	PositionArray:= GVL.aPosArray , 
	AxisGroupIdx:= GVL.nAxisIndex, 
	ExecuteCmd:= fbKRC_ReadTouchUPState.TouchUP OR GVL.HMI_TouchUpStoreNow, 
	Index:= , 
	Done=> , 
	Error=> , 
	ErrorID=> );

IF fbKRC_TouchUP.Done THEN
	fbKRC_TouchUP(ExecuteCmd := FALSE, PositionArray := GVL.aPosArray);
END_IF
END_ACTION

END_PROGRAM

// ---- POUs/mxAutomation/FB_AutoDemo.TcPOU
FUNCTION_BLOCK FB_AutoDemo
VAR_INPUT
	bExecute : BOOL;
END_VAR
VAR_OUTPUT
	bBusy : BOOL;
END_VAR
VAR
	nCurStep					: UDINT;
	i							: UDINT;
	nCurRunCount				: UDINT;
	fbMoveDirectAbs				: MC_MoveDirectAbsolute;
	fbMoveLinAbs 				: ARRAY [1..3] OF MC_MoveLinearAbsolute;
	fVeloM						: REAL := 2.0;
	fVeloPer					: REAL := 100.0;
	fAccM						: REAL := 2.3;
	fAccPer						: REAL := 100;
	
	stPrePos					: E6POS;
	stCoordSys					: COORDSYS;
	stApo1						: APO;
	
	fbKRC_Interrupt				: KRC_Interrupt;
	fbKRC_Continue				: KRC_Continue;
	
	iPosCount					: UINT :=1;
END_VAR
VAR CONSTANT
	POSARRLENGTH : UINT := 4;
END_VAR

CASE nCurStep OF
0:
	bBusy := FALSE;

	
	IF bExecute THEN
		iPosCount := 1;
		stApo1.CP_MODE := 0;
		stApo1.CDIS := 0;
		
		FOR i:= 1 TO 2  DO
			fbMoveLinAbs[i](Execute:= FALSE); 
		END_FOR
		fbMoveDirectAbs(Execute:= FALSE); 
		bBusy := TRUE;
		//PTP
		nCurStep := nCurStep + 10;
		nCurRunCount := 0;
		i := 0;
	END_IF
	
10:	
	M_MoveDirectToInitPos();
20:
	fbMoveLinAbs[2]();
	fbMoveLinAbs[3]();
	IF fbMoveLinAbs[1].ComAcpt AND NOT fbMoveLinAbs[2].Busy THEN
		fbMoveLinAbs[1].Execute := FALSE;
		iPosCount := iPosCount + 1;
		IF iPosCount > POSARRLENGTH THEN
			iPosCount := 1;
		END_IF
		nCurStep := nCurStep + 10;
	ELSE
		fbMoveLinAbs[1].Execute := TRUE;
	END_IF
	
	fbMoveLinAbs[1](
			AxisGroupIdx:= GVL.nAxisIndex, 
			Position:= GVL.aPosArray[iPosCount].E6POS, 
			Velocity:= fVeloM, 
			Acceleration:=fAccM , 
			CoordinateSystem:= stCoordSys, 
			OriType:= , 
			Approximate:= stApo1, 
			QueueMode:= 2 , 
			ComAcpt=> , 
			ComBusy=> , 
			Busy=> , 
			Active=> , 
			Done=> , 
			CommandAborted=> , 
			Error=> , 
			ErrorID=> );
		
		
	IF bExecute = FALSE THEN
		nCurStep := 100;
	END_IF

30:	
	fbMoveLinAbs[1]();
	fbMoveLinAbs[3]();
	
	IF fbMoveLinAbs[2].ComAcpt AND NOT fbMoveLinAbs[3].Busy THEN
		fbMoveLinAbs[2].Execute := FALSE;
		iPosCount := iPosCount + 1;
		IF iPosCount > POSARRLENGTH THEN
			iPosCount := 1;
		END_IF
		nCurStep := nCurStep + 10;
	ELSE
		fbMoveLinAbs[2].Execute := TRUE;
	END_IF	
	
	fbMoveLinAbs[2](
		AxisGroupIdx:= gvl.nAxisIndex, 
		Position:= GVL.aPosArray[iPosCount].E6POS, 
		Velocity:= fVeloM, 
		Acceleration:=fAccM , 
		CoordinateSystem:= stCoordSys, 
		OriType:= , 
		Approximate:= stApo1, 
		QueueMode:= 2 , 
		ComAcpt=> , 
		ComBusy=> , 
		Busy=> , 
		Active=> , 
		Done=> , 
		CommandAborted=> , 
		Error=> , 
		ErrorID=> );
		
	
	
	IF bExecute = FALSE THEN
		nCurStep := 100;
	END_IF
	
40:	
	fbMoveLinAbs[1]();
	fbMoveLinAbs[2]();
	
	IF fbMoveLinAbs[3].ComAcpt AND NOT fbMoveLinAbs[1].Busy THEN
		fbMoveLinAbs[3].Execute := FALSE;
		iPosCount := iPosCount + 1;
		IF iPosCount > POSARRLENGTH THEN
			iPosCount := 1;
		END_IF
		nCurStep := 20;
	ELSE
		fbMoveLinAbs[3].Execute := TRUE;
	END_IF	
	
	fbMoveLinAbs[3](
		AxisGroupIdx:= gvl.nAxisIndex, 
		Position:= GVL.aPosArray[iPosCount].E6POS, 
		Velocity:= fVeloM, 
		Acceleration:=fAccM , 
		CoordinateSystem:= stCoordSys, 
		OriType:= , 
		Approximate:= stApo1, 
		QueueMode:= 2 , 
		ComAcpt=> , 
		ComBusy=> , 
		Busy=> , 
		Active=> , 
		Done=> , 
		CommandAborted=> , 
		Error=> , 
		ErrorID=> );
		
	
	
	IF bExecute = FALSE THEN
		nCurStep := 100;
	END_IF
	
100:
	fbMoveLinAbs[1]();
	fbMoveLinAbs[2]();
	fbMoveLinAbs[3]();
	
	IF NOT bExecute AND NOT fbMoveDirectAbs.Busy 
		AND NOT fbMoveLinAbs[1].Busy AND NOT fbMoveLinAbs[2].Busy AND NOT fbMoveLinAbs[3].Busy THEN
		nCurStep := 0;
	END_IF
		
END_CASE

fbKRC_Interrupt(
	AxisGroupIdx:= GVL.nAxisIndex, 
	Execute:= , 
	Fast:= , 
	BrakeActive=> , 
	Error=> , 
	ErrorID=> );
	
fbKRC_Continue(AxisGroupIdx:= GVL.nAxisIndex, Enable:= , Error=> , ErrorID=> );

METHOD M_MoveDirectToInitPos : BOOL
VAR_INPUT
END_VAR
stPrePos := GVL.aPosArray[1].E6POS;
stCoordSys := GVL.aPosArray[1].COORDSYS;

fbMoveDirectAbs(
	AxisGroupIdx:= GVL.nAxisIndex , 
	Execute:= TRUE, 
	Position:= stPrePos, 
	Velocity:= fVeloPer , 
	Acceleration:=fAccPer , 
	CoordinateSystem:= stCoordSys , 
	Approximate:=stApo1 , 
	QueueMode:=  2, 
	ComAcpt=> , 
	ComBusy=> , 
	Busy=> , 
	Active=> , 
	Done=> , 
	CommandAborted=> , 
	Error=> , 
	ErrorID=> );
	
IF fbMoveDirectAbs.Done THEN
	fbMoveDirectAbs(Execute := FALSE); 
	nCurStep := nCurStep + 10;
END_IF
END_METHOD

END_FUNCTION_BLOCK

// ---- POUs/mxAutomation/Read_Axes_Velocity.TcPOU
PROGRAM Read_Axes_Velocity
VAR
	
	timer: Ton;
	
	// this function (ReadAxesVelocity) is an instance of the LIB (KRC_ReadActualAxisVelocity) function
	ReadAxesVelocity : KRC_ReadActualAxisVelocity;
	
	
	FLAG: BOOL;
	FLAG_Done: BOOL;
	VeloArray : ARRAY[1..6] OF INT;
	Read: BOOL;
END_VAR

	
	
timer(in:=NOT timer.q , PT:=T#100MS);
IF timer.Q THEN
	Read:=TRUE;
END_IF

///the function react only to rising edge of the INPPUT : ExecuteCmd
readaxesvelocity(
		axisgroupidx := gvl_settings.App_GroupIndex ,
		ExecuteCmd :=Read,
		done=> ,
		error=>,
		errorid=>,
		a1=> ,
		a2=> ,
		a3=> ,
		a4=> ,
		a5=> ,
		a6=> );

IF ReadAxesVelocity.Done  THEN
	FLAG_Done:=TRUE;
	Read:=FALSE;
	VeloArray[1]:=ReadAxesVelocity.A1;
	VeloArray[2]:=ReadAxesVelocity.A2;
	VeloArray[3]:=ReadAxesVelocity.A3;
	VeloArray[4]:=ReadAxesVelocity.A4;
	VeloArray[5]:=ReadAxesVelocity.A5;
	VeloArray[6]:=ReadAxesVelocity.A6;
ELSIF ReadAxesVelocity.Error THEN
	FLAG:=TRUE;
	Read:=FALSE;
END_IF
//END_IF

END_PROGRAM

// ---- POUs/CheckBounds.TcPOU
// Implicitly generated code : DO NOT EDIT
FUNCTION CheckBounds : DINT
VAR_INPUT
	index, lower, upper: DINT;
END_VAR
VAR_STAT
	counter:int;
END_VAR

// Implicitly generated code : Only an Implementation suggestion
{noflow}
IF  index < lower THEN
	CheckBounds := lower;
	counter:=counter+1;
ELSIF  index > upper THEN
	CheckBounds := upper;
	counter:=counter+1;
ELSE  
	CheckBounds := index;
END_IF
{flow}

END_FUNCTION

// ---- POUs/Prg_KillHMI.TcPOU
PROGRAM Prg_KillHMI
VAR
	fbKillHMI: NT_StartProcess;
	KillHMI:BOOL;
END_VAR


fbKillHMI(
	NETID:='' , 
	PATHSTR:='C:\TwinCAT\3.1\Boot\Plc\KillHMi_v2.bat' , 
	DIRNAME:='C:\TwinCAT\3.1\Boot\Plc' , 
	COMNDLINE:='' ,
	START:=KillHMI , 
	TMOUT:= T#10S, 
	BUSY=> , 
	ERR=> , 
	ERRID=> );	
KillHMI:=FALSE;

END_PROGRAM

// ---- POUs/Safety/FB_SafePower.TcPOU
// FB_SafePower sets contactor and lamp for one safety power output
FUNCTION_BLOCK FB_SafePower
VAR_INPUT
	bSwitchPower 		: BOOL; // switch is set to ON
	bHasPower			: BOOL; // contactor has power (Safety OK)
END_VAR
VAR_OUTPUT
	bLightSelectPower 	: BOOL; // lamp
	bSetSafetyPower		: BOOL; // bSwitchPower
END_VAR

VAR
//	fbBlink: FB_Blink;
END_VAR

bSetSafetyPower := bSwitchPower;

IF bSetSafetyPower AND bHasPower THEN
	bLightSelectPower := TRUE;
//ELSIF bSetSafetyPower AND NOT bHasPower THEN
//	fbBlink(bEnable:= TRUE, bOut=> bLightSelectPower);
ELSE
	bLightSelectPower := FALSE;
END_IF

END_FUNCTION_BLOCK

// ---- POUs/Safety/PRG_Safety.TcPOU
PROGRAM PRG_Safety
VAR
	fbRTrigGateRequest	: R_TRIG; //trigger for hw switch
	fbRTrigGateAck		: R_TRIG; //trigger for hw switch
//	fbBlinkGate			: fbBlinkGate;
	
	
	bGateAckSafety		: BOOL; //Resets and acknowledges all safety errors
	nStateSafetyReset	: UDINT;
	
	fbSafePower1		: FB_SafePower; //Sets lamp and unsafe power signal for power supply 1 
	fbSafePower2		: FB_SafePower; //Sets lamp and unsafe power signal for power supply 2
	tonSafetyGateAck	: TON :=(PT:=T#0.5S); //
	
	nZero: UDINT 		:= 0; // provoke division by 0 in case of fatal safety reset error
	bOut: BOOL;
END_VAR
VAR CONSTANT
	
END_VAR

//=====================================
//Power Kuka
//=====================================
GVL.out_DO2_1_Power230V_Kuka := GVL.in_DI1_3_SwitchPower3_230V;

GVL.out_DO1_3_LightSelectPower3 := GVL.in_DI1_3_SwitchPower3_230V;

//=====================================

//=====================================
// Gate 
//=====================================
fbRTrigGateRequest(CLK:=GVL.in_DI2_1_Tap_Request_SafetyGate);

IF fbRTrigGateRequest.Q THEN
	GVL.bToSafeGr1_GateRequest := TRUE;
	
	GVL.bToSafeGr1_ReqAutoMode := FALSE;
	
	bGateAckSafety := TRUE;
END_IF

fbRTrigGateAck(CLK:=GVL.in_DI2_2_AckSafetyGate);

IF fbRTrigGateAck.Q THEN
	GVL.bToSafeGr1_GateRequest := FALSE; 
	GVL.bToSafeGr1_ReqAutoMode := TRUE;
	bGateAckSafety := TRUE;
END_IF

//=====================================


//=====================================
// Gate Lamps
//=====================================
IF GVL.bFromSafeGr1_GateUnlocked THEN
	
	GVL.out_DO1_5_LightReqSafetyGate := TRUE;
	GVL.out_DO1_6_LightAckSafetyGate := FALSE;
ELSIF GVL.bFromSafeGr1_Power THEN
	GVL.out_DO1_5_LightReqSafetyGate := FALSE;
	GVL.out_DO1_6_LightAckSafetyGate := TRUE;
ELSIF GVL.bToSafeGr1_GateRequest THEN
//	fbBlinkGate(bEnable:= TRUE);
//	GVL.out_DO1_5_LightReqSafetyGate := fbBlinkGate.bOut;
	GVL.out_DO1_6_LightAckSafetyGate := FALSE;
ELSIF GVL.bToSafeGr1_ReqAutoMode THEN
//	fbBlinkGate(bEnable:= TRUE);
	GVL.out_DO1_5_LightReqSafetyGate := FALSE;
//	GVL.out_DO1_6_LightAckSafetyGate := fbBlinkGate.bOut;
ELSE
	gvl.out_DO1_5_LightReqSafetyGate := FALSE;
	gvl.out_DO1_5_LightReqSafetyGate := FALSE;
END_IF
//=====================================


//=====================================
// Safety Confirmation/Reset
// Called to start automatic mode
//=====================================

CASE nStateSafetyReset OF
0:  
	IF bGateAckSafety THEN
		nStateSafetyReset := nStateSafetyReset + 10;
	END_IF
10:
	GVL.bToSafeGr1_RunStopGrp1 := TRUE;
	
	nStateSafetyReset := nStateSafetyReset + 10;
20:
	GVL.bToSafeGr1_ErrAck := TRUE;
	
	GVL.bToSafeGr2_ErrAck := TRUE;
	
	
	IF GVL.bToSafeGr1_ReqAutoMode THEN
		nStateSafetyReset := 110;
	ELSE
		nStateSafetyReset := nStateSafetyReset := 500; //end
	END_IF
110:	// following steps may only be run if auto mode is requested

	GVL.bToSafeGr1_EStopRestart1 := TRUE;
	
	GVL.bToSafeGr1_EStopRestart2 := TRUE;
	
	nStateSafetyReset := nStateSafetyReset + 10;
120:
	GVL.bToSafeGr1_GateMonReset := TRUE;
	
	nStateSafetyReset := nStateSafetyReset + 10;

130:
	//falling edge for reset 
	tonSafetyGateAck(IN:= TRUE, PT := T#0.5S);
	IF tonSafetyGateAck.Q THEN
		tonSafetyGateAck(IN:= FALSE, PT := T#0.5S);
		GVL.bToSafeGr1_GateMonReset := FALSE;
		nStateSafetyReset := 500;
	END_IF
500:

	GVL.bToSafeGr1_ErrAck := FALSE;
	GVL.bToSafeGr2_ErrAck := FALSE;
	GVL.bToSafeGr1_EStopRestart1 := FALSE;
	GVL.bToSafeGr1_EStopRestart2 := FALSE;
	GVL.bToSafeGr1_GateMonReset := FALSE;
	bGateAckSafety := FALSE;
	
	IF NOT bGateAckSafety THEN
		nStateSafetyReset := 0;
	END_IF
END_CASE

//provoke division by 0 if auto mode is reset while auto mode not required
IF ((NOT GVL.bToSafeGr1_ReqAutoMode) AND nStateSafetyReset >= 100 AND nStateSafetyReset < 500) THEN 
	nStateSafetyReset := 0/nZero;
END_IF
//=====================================

//=====================================
// Power switches
//=====================================
fbSafePower1(bSwitchPower:= GVL.in_DI1_1_SwitchPower1_230V, bHasPower:= GVL.bFromSafeGr1_Power1_230V , bLightSelectPower=> GVL.out_DO1_1_LightSelectPower1, bSetSafetyPower=> GVL.bToSafeGr1_Power1_230V);
fbSafePower2(bSwitchPower:= GVL.in_DI1_2_SwitchPower2_230V, bHasPower:= GVL.bFromSafeGr1_Power2_230V , bLightSelectPower=> GVL.out_DO1_2_LightSelectPower2, bSetSafetyPower=> GVL.bToSafeGr1_Power2_230V);
//=====================================

END_PROGRAM

// ---- GlobalTextList.TcGTLO
TEXTLIST GlobalTextList
  1920 = ''
  1111 = ' controller ready for\nstart'
  83 = ' controller ready for program\nstart'
  63 = ' controller ready for start'
  380 = ' mode T1 selected'
  1590 = ' mode T2 selected'
  773 = ' stop by E.\nSTOP'
  1354 = ' stop by E.STOP'
  593 = ' stop by EMERGENCY\nSTOP'
  1725 = '%.2f'
  1 = '%d'
  437 = '%D'
  309 = '%s'
  1879 = "'DIAGNOSTIC' error"
  807 = "'ERROR' error"
  8 = '+   A1 / X '
  13 = '+   A2 / Y '
  15 = '+   A3 / Z '
  17 = '+   A4 / A '
  19 = '+   A5 / B '
  21 = '+   A6 / C '
  9 = '-   A1 / X '
  14 = '-   A2 / Y '
  16 = '-   A3 / Z '
  18 = '-   A4 / A '
  20 = '-   A5 / B '
  22 = '-   A6 / C '
  12 = '0-PTP axial 1-LIN cart 2-SPTP 3-SLIN'
  615 = '1234567890'
  32 = 'A'
  624 = 'a'
  38 = 'A1'
  620 = 'a1'
  137 = 'A1Label'
  39 = 'A2'
  71 = 'a2'
  1501 = 'A2A2'
  110 = 'A2Label'
  40 = 'A3'
  655 = 'a3'
  41 = 'A4'
  775 = 'a4'
  42 = 'A5'
  376 = 'a5'
  43 = 'A6'
  87 = 'a6'
  2300 = 'AAPPROACH'
  553 = 'acceleration'
  1228 = 'acknolage'
  1330 = 'acknowledge'
  1517 = 'Aes Velocityon'
  407 = 'alarm stop'
  914 = 'appl run'
  408 = 'APPROACH'
  1652 = 'AUTO EXT \nactive'
  449 = 'auto ext \nactive'
  544 = 'AUTO EXT  active'
  85 = 'AUTO EXT  I/F active'
  1324 = 'auto ext active'
  1978 = 'Auto ext I/F active'
  1487 = 'auto external  I/F active'
  274 = 'Automat'
  50 = 'Automatic'
  52 = 'Automatic Continue'
  53 = 'Automatic External'
  1564 = 'Automatic External \nactive'
  1326 = 'Automatic External interface\nactive'
  51 = 'Automatic Interrupt'
  3 = 'AutoStart'
  334 = 'Axes Motion'
  1125 = 'Axes Position'
  1989 = 'axes software imits'
  1121 = 'Axes SW limits'
  2274 = 'Axes Velocity'
  33 = 'B'
  6 = 'BASE %d'
  34 = 'C'
  187 = 'communication'
  345 = 'Communication'
  59 = 'Connect'
  382 = 'Continue'
  809 = 'Coordinate System'
  1299 = 'Diag Err'
  458 = 'diagnosis'
  790 = 'diagnostic'
  764 = 'done'
  1990 = 'DONE'
  61 = 'drives not ready'
  943 = 'Drives Off'
  893 = 'drives off'
  76 = 'enable AUTO'
  678 = 'Enable Automat'
  1861 = 'enable automat'
  57 = 'Enable External'
  64 = 'enable external'
  373 = 'Enable T1'
  1534 = 'enable T1'
  350 = 'Enable T2'
  1180 = 'enable T2'
  741 = 'erro'
  160 = 'ERROR'
  1188 = 'error'
  676 = 'Error'
  28 = 'Error %d'
  664 = 'Error err'
  307 = 'error ID'
  778 = 'Error Number'
  1023 = 'errorID'
  560 = 'EXIT'
  27 = 'EXT'
  1453 = 'ext I/F active'
  1182 = 'EXT mode'
  56 = 'External'
  2163 = 'EXTERNAL mode'
  1614 = 'FOLD'
  77 = 'General settings'
  490 = 'GO'
  931 = 'gO lINEAR'
  692 = 'Go To %s'
  37 = 'GVL.HMI_ActualCartPos.E5'
  609 = 'heaertbit PNOS'
  964 = 'Heartbit KRC'
  926 = 'heartbitPNOS'
  498 = 'HOME'
  129 = 'home'
  797 = 'homeLabel'
  25 = 'I'
  48 = 'in LIN motion'
  49 = 'in PTP motion'
  1015 = 'Init Error'
  360 = 'Init Error numbe'
  548 = 'Init Error number'
  58 = 'Initialize'
  68 = 'int e stop'
  1335 = 'internal E stop'
  430 = 'IO act conf'
  7 = 'JOG- Mode: %d'
  1767 = 'KRC error'
  1256 = 'KRC error Active'
  574 = 'KRC errorACtive'
  60 = 'KRC errorActive'
  285 = 'Label'
  11 = 'Load %d kg'
  878 = 'MAIN'
  1142 = 'MAINTENANCE'
  994 = 'message'
  1368 = 'Message Count'
  2130 = 'Message Countaxes mastered'
  578 = 'Mode'
  1239 = 'mode AUTO selected'
  1157 = 'mode EXTERNAL selected'
  1225 = 'Motion Axes'
  786 = 'motion command'
  798 = 'Motion Command'
  162 = 'motion feedback'
  159 = 'Motion Feedback'
  1947 = 'Motion lINEAR'
  2301 = 'Motion Linear'
  976 = 'Motion Linear ,move tool in linear path'
  2144 = 'MotionAxes'
  219 = 'Move Enable'
  984 = 'move enable'
  47 = 'Move to Position %d'
  948 = 'mxA_Motion.fbKRC_ReadActualPosition.Position'
  1875 = 'mxA_Motion.fbKRC_ReadActualPosition.Position.A'
  1884 = 'mxA_Motion.fbKRC_ReadActualPosition.Position.B'
  1893 = 'mxA_Motion.fbKRC_ReadActualPosition.Position.C'
  1902 = 'mxA_Motion.fbKRC_ReadActualPosition.Position.Status'
  1911 = 'mxA_Motion.fbKRC_ReadActualPosition.Position.Turn'
  1848 = 'mxA_Motion.fbKRC_ReadActualPosition.Position.X'
  1857 = 'mxA_Motion.fbKRC_ReadActualPosition.Position.Y'
  1866 = 'mxA_Motion.fbKRC_ReadActualPosition.Position.Z'
  944 = 'near pos ret'
  98 = 'ner pos ret'
  1131 = 'no Heart bit KRC'
  228 = 'no heartbit PNOS'
  1279 = 'no heartbitPNOS'
  706 = 'no MOVE enable'
  1193 = 'no OP Mode EXT'
  1000 = 'no prog active'
  1198 = 'not INIT'
  1150 = 'not on line'
  284 = 'on path'
  1389 = 'op mode AUTO selected'
  898 = 'op mode EXTERNAL selected'
  595 = 'op mode T1 selected'
  216 = 'op mode T2 selected'
  1018 = 'operating mode T1 selected'
  1484 = 'operator safety violated'
  117 = 'ORIGIN'
  2 = 'Override'
  640 = 'Override Speed'
  1076 = 'override speed : %d'
  24 = 'P'
  1398 = 'Pause'
  123 = 'pery ready'
  45 = 'Position in Array %d'
  55 = 'pro act'
  346 = 'pro move'
  817 = 'process active at robot level'
  26 = 'R'
  54 = 'RC ready'
  1771 = 'READ '
  214 = 'Read KRC error'
  2677 = 'Read_Axes_Velocity.ReadAxesVelocity.AxisGroupIdx'
  2696 = 'Read_Axes_Velocity.ReadAxesVelocity.Done'
  2705 = 'Read_Axes_Velocity.ReadAxesVelocity.Error'
  2715 = 'Read_Axes_Velocity.ReadAxesVelocity.ErrorID'
  2686 = 'Read_Axes_Velocity.ReadAxesVelocity.ExecuteCmd'
  2277 = 'RESET'
  1510 = 'Reset'
  539 = 'reset auto eext'
  226 = 'reset auto external'
  44 = 'Reset AutoExt'
  1689 = 'reset message'
  4 = 'Reset messages'
  1038 = 'restart'
  662 = 'rob stopped'
  1527 = 'robot axes mastered'
  509 = 'robot cal'
  1277 = 'robot controller ready for program\nstart'
  62 = 'robot drives activated'
  128 = 'Robot FW major'
  82 = 'Robot FW minor'
  263 = 'Robot FW revision'
  799 = 'Robot FW version'
  1417 = 'robot is at standstill'
  642 = 'robot near saved position'
  1408 = 'robot on programmed path'
  1297 = 'robot program running'
  333 = 'Robot Serial'
  421 = 'robot stop by EMERGENCY\nSTOP'
  306 = 'robot stopped'
  720 = 'run'
  370 = 'Rx'
  1253 = 'Ry'
  1500 = 'Rz'
  23 = 'S'
  641 = 'safe not OK'
  1213 = 'safety'
  1291 = 'safety circuit interrupted'
  840 = 'Safety Communication'
  1404 = 'Safety interuption'
  0 = 'Safety-Rese'
  830 = 'Serial'
  511 = 'settings'
  2225 = 'shavouot'
  540 = 'Speed'
  35 = 'Status'
  282 = 'status'
  96 = 'stop mess'
  1351 = 'STOPMESS'
  46 = 'Store ->'
  710 = 'synchronous motion active'
  572 = 'synchronous robot active'
  796 = 'synchronous robot motion active'
  436 = 'T1 '
  182 = 'T2'
  894 = 'target'
  1122 = 'Target Command'
  497 = 'time : '
  5 = 'TOOL %d'
  668 = 'tool poian coordinate system'
  163 = 'tool position'
  1795 = 'Tool Position'
  648 = 'tool position , tool tip position in Cartesian coordinate system'
  269 = 'Toool Number'
  584 = 'Traget Position'
  36 = 'Turn'
  1273 = 'turn'
  148 = 'user safe'
  145 = 'user safe not ok'
  771 = 'velocity'
  549 = 'Win Counter'
  494 = 'win OS counter'
  438 = 'Windows Counter'
  699 = 'windows counter'
  279 = 'Windows Counter :'
  802 = 'windows time'
  10 = 'Write Load Data'
  29 = 'X'
  550 = 'x'
  1577 = 'xA1'
  30 = 'Y'
  1796 = 'y'
  31 = 'Z'
  2035 = 'z'
END_TEXTLIST

// ---- VISUs/APP_Settings.TcVIS
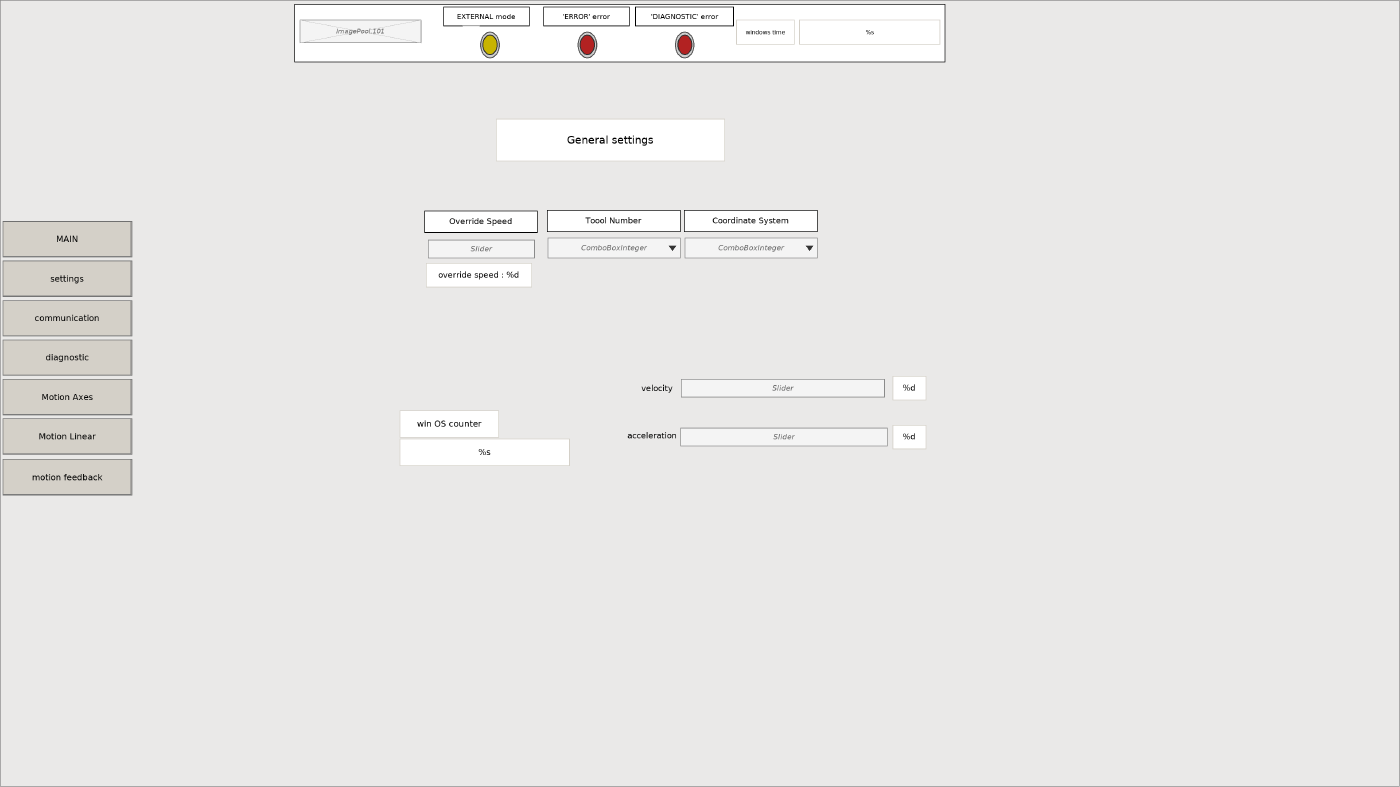
VISUALIZATION APP_Settings  // 1920x1080
    Frame (400,1 900x90)
        shows MenuTop()
    Frame (0,300 200x400)
        shows MenuMain()
    Textfield (680,163 314x58), "General settings"
    Rectangle (582,289 155x30), "Override Speed"
    Rectangle (750,288 183x30), "Toool Number"
    ComboBoxInteger (751,326 182x28), variable: GVL_settings.App_CoordSys.TOOL, text list: 'ToolNumber'
    Slider (934,520 279x25), variable: GVL_settings.App_Velocity, scale 10..50
    Slider (933,587 284x25), variable: GVL_settings.App_Acceleration, scale 10..50
    Label (865,519 72x28), "velocity"
    Label (849,584 91x28), "acceleration"
    Textfield (1224,516 46x33), "%d", text variable: GVL_settings.App_Velocity
    Textfield (1224,583 46x33), "%d", text variable: GVL_settings.App_Acceleration
    Textfield (548,563 136x37), "win OS counter"
    Textfield (548,602 233x37), "%s", text variable: GVL_PLC.Str_windowsCounter
    Rectangle (938,288 183x30), "Coordinate System"
    ComboBoxInteger (939,326 182x28), variable: GVL_settings.App_CoordSys.BASE, text list: 'CoorSys'
    Slider (587,329 146x25), variable: GVL.nOverrideGlobal, scale 10..50
    Textfield (584,361 145x33), "override speed : %d", text variable: GVL.nOverrideGlobal
END_VISUALIZATION

// ---- VISUs/diagnostic.TcVIS
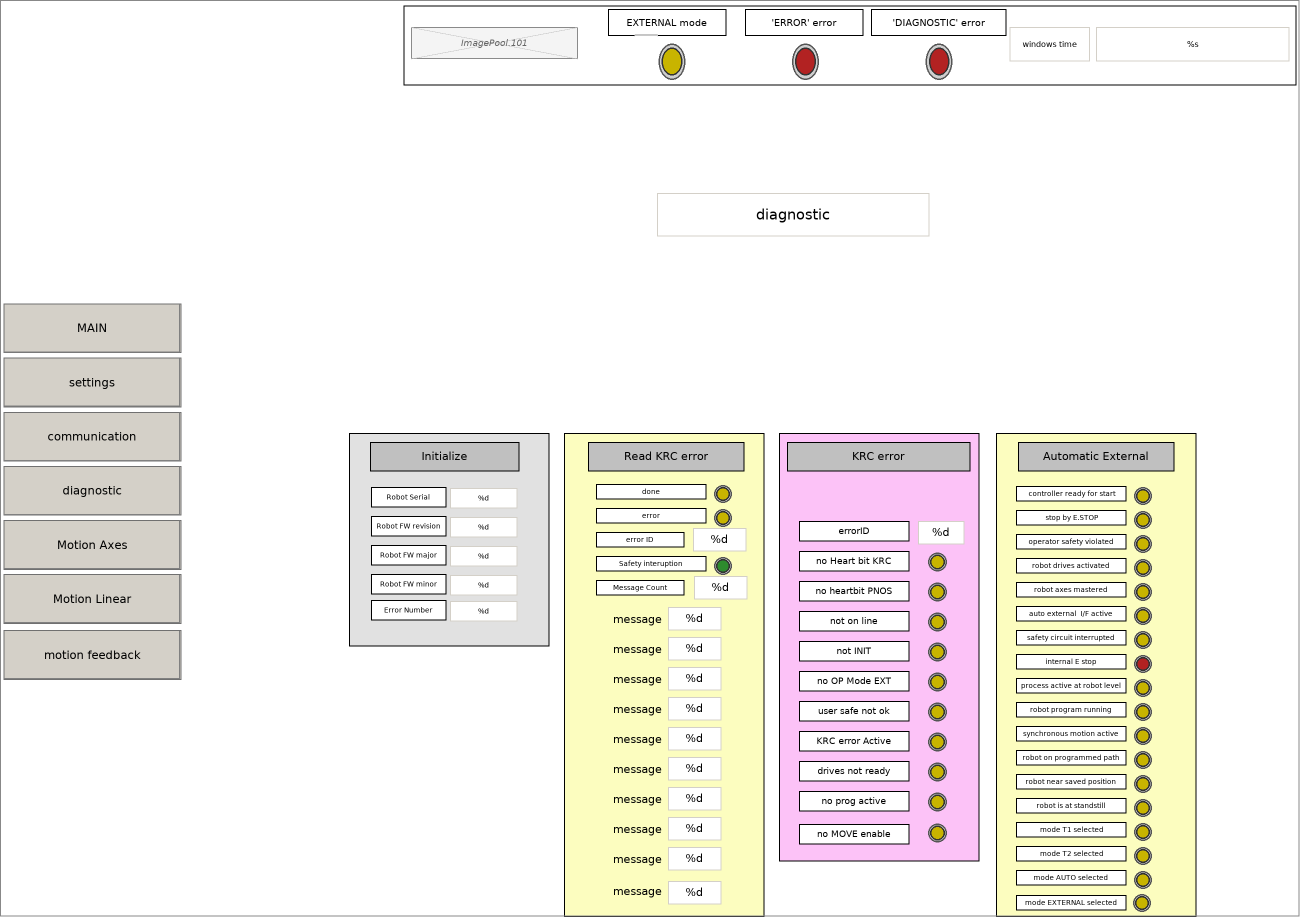
VISUALIZATION diagnostic  // 1300x917
    Rectangle (996,433 200x484), text variable: MAIN.fbKRC_Error.ErrorID
    Rectangle (349,433 200x213)
    Rectangle (779,433 200x428)
    Frame (400,1 900x90)
        shows MenuTop()
    Frame (0,300 200x400)
        shows MenuMain()
    Textfield (657,193 272x43), "diagnostic"
    Lamp1 (1123,486 40x20), variable: MAIN.fbKRC_AutomaticExternal.RC_RDY1, style: Lamp-Lamp1-Yellow
    Lamp1 (1123,510 40x20), variable: MAIN.fbKRC_AutomaticExternal.ALARM_STOP, style: Lamp-Lamp1-Yellow
    Lamp1 (1123,534 40x20), variable: MAIN.fbKRC_AutomaticExternal.USER_SAFE, style: Lamp-Lamp1-Yellow
    Lamp1 (1123,558 40x20), variable: MAIN.fbKRC_AutomaticExternal.PERI_RDY, style: Lamp-Lamp1-Yellow
    Lamp1 (1123,582 40x20), variable: MAIN.fbKRC_AutomaticExternal.ROB_CAL, style: Lamp-Lamp1-Yellow
    Lamp1 (1123,606 40x20), variable: MAIN.fbKRC_AutomaticExternal.IO_ACTCONF, style: Lamp-Lamp1-Yellow
    Rectangle (371,516 75x20), "Robot FW revision"
    Rectangle (371,545 75x20), "Robot FW major"
    Rectangle (371,574 75x20), "Robot FW minor"
    Textfield (450,517 67x20), "%d", text variable: MAIN.fbKRC_Initialize.KRC_Revision
    Textfield (450,546 67x20), "%d", text variable: MAIN.fbKRC_Initialize.KRC_Major
    Textfield (450,575 67x20), "%d", text variable: MAIN.fbKRC_Initialize.KRC_Minor
    Rectangle (371,487 75x20), "Robot Serial"
    Textfield (450,488 67x20), "%d", text variable: MAIN.fbKRC_Initialize.KRC_Serial
    Rectangle (1018,442 156x29), "Automatic External", text variable: GVL.HMI_Error_General_ID, colour toggle: GVL.HMI_Error_General
    Rectangle (1016,486 110x15), "controller ready for start", text variable: GVL.HMI_Error_General_ID, colour toggle: GVL.HMI_Error_General
    Rectangle (1016,510 110x15), "stop by E.STOP", text variable: GVL.HMI_Error_General_ID, colour toggle: GVL.HMI_Error_General
    Rectangle (1016,534 110x15), "operator safety violated", text variable: GVL.HMI_Error_General_ID, colour toggle: GVL.HMI_Error_General
    Rectangle (1016,558 110x15), "robot drives activated", text variable: GVL.HMI_Error_General_ID, colour toggle: GVL.HMI_Error_General
    Rectangle (1016,582 110x15), "robot axes mastered", text variable: GVL.HMI_Error_General_ID, colour toggle: GVL.HMI_Error_General
    Rectangle (1016,606 110x15), "auto external I/F active", text variable: GVL.HMI_Error_General_ID, colour toggle: GVL.HMI_Error_General
    Lamp1 (1123,630 40x20), variable: MAIN.fbKRC_AutomaticExternal.STOPMESS, style: Lamp-Lamp1-Yellow
    Lamp1 (1123,654 40x20), variable: MAIN.NOT_INT_E_STOP, style: Lamp-Lamp1-Red
    Lamp1 (1123,678 40x20), variable: MAIN.fbKRC_AutomaticExternal.PRO_ACT, style: Lamp-Lamp1-Yellow
    Rectangle (1016,630 110x15), "safety circuit interrupted", text variable: GVL.HMI_Error_General_ID, colour toggle: GVL.HMI_Error_General
    Rectangle (1016,654 110x15), "internal E stop", text variable: GVL.HMI_Error_General_ID, colour toggle: GVL.HMI_Error_General
    Rectangle (1016,678 110x15), "process active at robot level", text variable: GVL.HMI_Error_General_ID, colour toggle: GVL.HMI_Error_General
    Lamp1 (1123,702 40x20), variable: MAIN.fbKRC_AutomaticExternal.APPL_RUN, style: Lamp-Lamp1-Yellow
    Rectangle (1016,702 110x15), "robot program running", text variable: GVL.HMI_Error_General_ID, colour toggle: GVL.HMI_Error_General
    Lamp1 (1123,726 40x20), variable: MAIN.fbKRC_AutomaticExternal.PRO_MOVE, style: Lamp-Lamp1-Yellow
    Lamp1 (1123,750 40x20), variable: MAIN.fbKRC_AutomaticExternal.ON_PATH, style: Lamp-Lamp1-Yellow
    Lamp1 (1123,774 40x20), variable: MAIN.fbKRC_AutomaticExternal.NEAR_POSRET, style: Lamp-Lamp1-Yellow
    Rectangle (1016,726 110x15), "synchronous motion active", text variable: GVL.HMI_Error_General_ID, colour toggle: GVL.HMI_Error_General
    Rectangle (1016,750 110x15), "robot on programmed path", text variable: GVL.HMI_Error_General_ID, colour toggle: GVL.HMI_Error_General
    Rectangle (1016,774 110x15), "robot near saved position", text variable: GVL.HMI_Error_General_ID, colour toggle: GVL.HMI_Error_General
    Rectangle (1016,798 110x15), "robot is at standstill", text variable: GVL.HMI_Error_General_ID, colour toggle: GVL.HMI_Error_General
    Rectangle (1016,822 110x15), "mode T1 selected", text variable: GVL.HMI_Error_General_ID, colour toggle: GVL.HMI_Error_General
    Rectangle (1016,846 110x15), "mode T2 selected", text variable: GVL.HMI_Error_General_ID, colour toggle: GVL.HMI_Error_General
    Rectangle (1016,870 110x15), "mode AUTO selected", text variable: GVL.HMI_Error_General_ID, colour toggle: GVL.HMI_Error_General
    Rectangle (1016,895 110x15), "mode EXTERNAL selected", text variable: GVL.HMI_Error_General_ID, colour toggle: GVL.HMI_Error_General
    Lamp1 (1123,798 40x20), variable: MAIN.fbKRC_AutomaticExternal.PRO_ACT, style: Lamp-Lamp1-Yellow
    Lamp1 (1123,822 40x20), variable: MAIN.fbKRC_AutomaticExternal.T1, style: Lamp-Lamp1-Yellow
    Lamp1 (1123,846 40x20), variable: MAIN.fbKRC_AutomaticExternal.T2, style: Lamp-Lamp1-Yellow
    Lamp1 (1123,870 40x20), variable: MAIN.fbKRC_AutomaticExternal.AUT, style: Lamp-Lamp1-Yellow
    Lamp1 (1123,893 38x20), variable: MAIN.fbKRC_AutomaticExternal.EXT, style: Lamp-Lamp1-Yellow
    Rectangle (370,442 149x29), "Initialize", text variable: GVL.HMI_Error_General_ID, colour toggle: GVL.HMI_Error_General
    Rectangle (371,600 75x20), "Error Number"
    Textfield (450,601 67x20), "%d", text variable: MAIN.fbKRC_Initialize.Error
    Rectangle (787,442 183x29), "KRC error", text variable: GVL.HMI_Error_General_ID, colour toggle: GVL.HMI_Error_General
    Rectangle (799,521 110x20), "errorID"
    Rectangle (799,551 110x20), "no Heart bit KRC"
    Rectangle (799,581 110x20), "no heartbit PNOS"
    Rectangle (799,611 110x20), "not on line"
    Rectangle (799,641 110x20), "not INIT"
    Rectangle (799,671 110x20), "no OP Mode EXT"
    Rectangle (799,701 110x20), "user safe not ok"
    Rectangle (799,731 110x20), "KRC error Active"
    Rectangle (799,761 110x20), "drives not ready"
    Rectangle (799,791 110x20), "no prog active"
    Rectangle (799,824 110x20), "no MOVE enable"
    Lamp1 (926,551 23x22), variable: MAIN.fbKRC_Error.NoHeartbeatKRC, style: Lamp-Lamp1-Yellow
    Lamp1 (926,581 23x22), variable: MAIN.fbKRC_Error.NoHeartbeatPCOS, style: Lamp-Lamp1-Yellow
    Lamp1 (926,611 23x22), variable: MAIN.fbKRC_Error.NoMoveEnable, style: Lamp-Lamp1-Yellow
    Lamp1 (926,641 23x22), variable: MAIN.fbKRC_Error.NotInitialized, style: Lamp-Lamp1-Yellow
    Lamp1 (926,671 23x22), variable: MAIN.fbKRC_Error.NoOpModeExt, style: Lamp-Lamp1-Yellow
    Lamp1 (926,701 23x22), variable: MAIN.fbKRC_Error.UserSafeNotOK, style: Lamp-Lamp1-Yellow
    Lamp1 (926,731 23x22), variable: MAIN.fbKRC_Error.KrcErrorActive, style: Lamp-Lamp1-Yellow
    Lamp1 (926,761 23x22), variable: MAIN.fbKRC_Error.DrivesNotReady, style: Lamp-Lamp1-Yellow
    Lamp1 (926,791 23x22), variable: MAIN.fbKRC_Error.NoProgActive, style: Lamp-Lamp1-Yellow
    Lamp1 (926,822 23x22), variable: MAIN.fbKRC_Error.NoMoveEnable, style: Lamp-Lamp1-Yellow
    Textfield (918,521 46x23), "%d", text variable: MAIN.fbKRC_Error.ErrorID
    Rectangle (564,433 200x484), text variable: MAIN.fbKRC_Error.ErrorID
    Lamp1 (703,484 40x20), variable: MAIN.ReadKRCError.Done, style: Lamp-Lamp1-Yellow
    Lamp1 (703,508 40x20), variable: MAIN.ReadKRCError.Error, style: Lamp-Lamp1-Yellow
    Lamp1 (703,556 40x20), variable: NOT(MAIN.ReadKRCError.STOPMESS), style: Lamp-Lamp1-Green
    Rectangle (588,442 156x29), "Read KRC error", text variable: GVL.HMI_Error_General_ID, colour toggle: GVL.HMI_Error_General
    Rectangle (596,484 110x15), "done", text variable: GVL.HMI_Error_General_ID, colour toggle: GVL.HMI_Error_General
    Rectangle (596,508 110x15), "error", text variable: GVL.HMI_Error_General_ID, colour toggle: GVL.HMI_Error_General
    Rectangle (596,532 88x15), "error ID", text variable: GVL.HMI_Error_General_ID, colour toggle: GVL.HMI_Error_General
    Rectangle (596,556 110x15), "Safety interuption", text variable: MAIN.ReadKRCError.STOPMESS, colour toggle: GVL.HMI_Error_General
    Rectangle (596,580 88x15), "Message Count", text variable: GVL.HMI_Error_General_ID, colour toggle: GVL.HMI_Error_General
    Textfield (693,528 53x23), "%d", text variable: MAIN.ReadKRCError.ErrorID
    Textfield (694,576 53x23), "%d", text variable: MAIN.ReadKRCError.ErrorID
    Textfield (668,607 53x23), "%d", text variable: MAIN.ReadKRCError.Message1
    Textfield (668,637 53x23), "%d", text variable: MAIN.ReadKRCError.Message2
    Textfield (668,667 53x23), "%d", text variable: MAIN.ReadKRCError.Message3
    Textfield (668,697 53x23), "%d", text variable: MAIN.ReadKRCError.Message4
    Textfield (668,727 53x23), "%d", text variable: MAIN.ReadKRCError.Message5
    Textfield (668,757 53x23), "%d", text variable: MAIN.ReadKRCError.Message6
    Textfield (668,787 53x23), "%d", text variable: MAIN.ReadKRCError.Message7
    Textfield (668,817 53x23), "%d", text variable: MAIN.ReadKRCError.Message8
    Textfield (668,847 53x23), "%d", text variable: MAIN.ReadKRCError.Message9
    Textfield (668,881 53x23), "%d", text variable: MAIN.ReadKRCError.Message10
    Label (612,605 51x29), "message"
    Label (612,635 51x29), "message"
    Label (612,665 51x29), "message"
    Label (612,695 51x29), "message"
    Label (612,725 51x29), "message"
    Label (612,755 51x29), "message"
    Label (612,785 51x29), "message"
    Label (612,815 51x29), "message"
    Label (612,845 51x29), "message"
    Label (612,877 51x29), "message"
END_VISUALIZATION

// ---- VISUs/communication.TcVIS
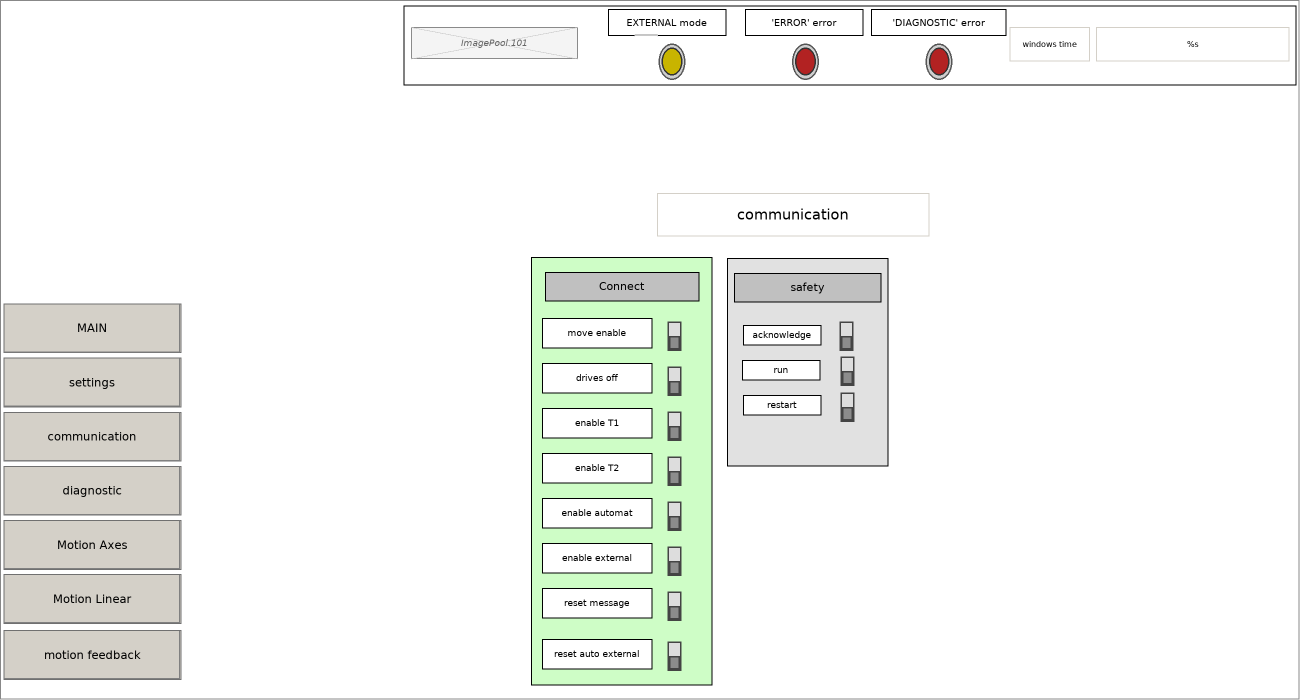
VISUALIZATION communication  // 1300x700
    Rectangle (531,257 181x428)
    Frame (400,1 900x90)
        shows MenuTop()
    Frame (0,300 200x400)
        shows MenuMain()
    Textfield (657,193 272x43), "communication"
    Rectangle (545,272 154x29), "Connect", text variable: GVL.HMI_Error_General_ID, colour toggle: GVL.HMI_Error_General
    DipSwitch (660,316 29x40), variable: MAIN.fbKRC_AutomaticExternal.MOVE_ENABLE, behaviour: TOGGLE, style: Switch-DipSwitch-Gray
    DipSwitch (660,361 29x40), variable: MAIN.fbKRC_AutomaticExternal.DRIVES_OFF, behaviour: TOGGLE, style: Switch-DipSwitch-Gray
    DipSwitch (660,406 29x40), variable: MAIN.fbKRC_AutomaticExternal.ENABLE_T1, behaviour: TOGGLE, style: Switch-DipSwitch-Gray
    DipSwitch (660,451 29x40), variable: MAIN.fbKRC_AutomaticExternal.ENABLE_T2, behaviour: TOGGLE, style: Switch-DipSwitch-Gray
    DipSwitch (660,496 29x40), variable: MAIN.fbKRC_AutomaticExternal.ENABLE_AUT, behaviour: TOGGLE, style: Switch-DipSwitch-Gray
    DipSwitch (660,541 29x40), variable: MAIN.fbKRC_AutomaticExternal.ENABLE_EXT, behaviour: TOGGLE, style: Switch-DipSwitch-Gray
    DipSwitch (660,586 29x40), variable: MAIN.fbKRC_Error.MessageReset, behaviour: TOGGLE, style: Switch-DipSwitch-Gray
    DipSwitch (660,636 29x40), variable: MAIN.fbKRC_AutomaticExternal.RESET, behaviour: TOGGLE, style: Switch-DipSwitch-Gray
    Rectangle (727,258 161x208)
    Rectangle (734,273 147x29), "safety", text variable: GVL.HMI_Error_General_ID, colour toggle: GVL.HMI_Error_General
    DipSwitch (832,316 29x40), variable: GVL_SAFETY.Ack, behaviour: TOGGLE, style: Switch-DipSwitch-Gray
    DipSwitch (833,351 29x40), variable: GVL_SAFETY.Run, behaviour: TOGGLE, style: Switch-DipSwitch-Gray
    DipSwitch (833,387 29x40), variable: GVL_SAFETY.Restart, behaviour: TOGGLE, style: Switch-DipSwitch-Gray
    Rectangle (743,325 78x20), "acknowledge"
    Rectangle (742,360 78x20), "run"
    Rectangle (743,395 78x20), "restart"
    Rectangle (542,318 110x30), "move enable"
    Rectangle (542,363 110x30), "drives off"
    Rectangle (542,408 110x30), "enable T1"
    Rectangle (542,453 110x30), "enable T2"
    Rectangle (542,498 110x30), "enable automat"
    Rectangle (542,543 110x30), "enable external"
    Rectangle (542,588 110x30), "reset message"
    Rectangle (542,639 110x30), "reset auto external"
END_VISUALIZATION

// ---- VISUs/Motion_Axes.TcVIS
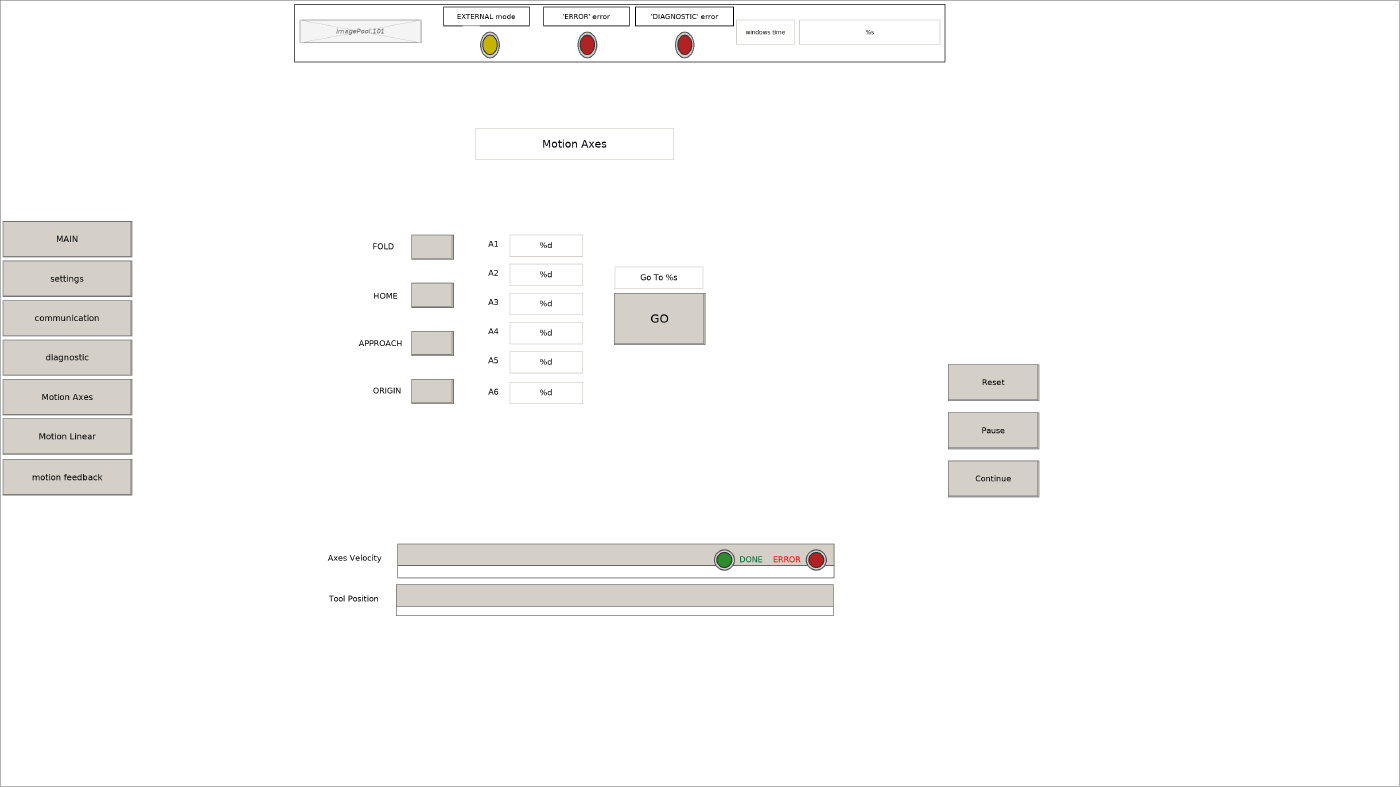
VISUALIZATION Motion_Axes  // 1920x1080
    Frame (400,1 900x90)
        shows MenuTop()
    Frame (0,300 200x400)
        shows MenuMain()
    Textfield (652,176 272x43), "Motion Axes"
    Button (1300,566 125x50), "Pause"
        tap mxA_Motion.fbAutoDemo.fbKRC_Interrupt.Execute
    Button (1300,632 125x50), "Continue"
        tap mxA_Motion.fbAutoDemo.fbKRC_Continue.Enable
    Button (842,402 125x71), "GO"
        tap MAIN.Move_Axes.Execute
    Textfield (699,322 100x30), "%d", text variable: MAIN.Move_Axes.AxisPosition.A1
    Textfield (699,362 100x30), "%d", text variable: MAIN.Move_Axes.AxisPosition.A2
    Textfield (699,402 100x30), "%d", text variable: MAIN.Move_Axes.AxisPosition.A3
    Textfield (699,442 100x30), "%d", text variable: MAIN.Move_Axes.AxisPosition.A4
    Textfield (699,482 100x30), "%d", text variable: MAIN.Move_Axes.AxisPosition.A5
    Textfield (699,524 100x30), "%d", text variable: MAIN.Move_Axes.AxisPosition.A6
    Label (660,323 34x24), "A1"
    Label (660,363 34x24), "A2"
    Label (660,403 34x24), "A3"
    Label (660,443 34x24), "A4"
    Label (660,483 34x24), "A5"
    Label (660,526 34x24), "A6"
    Button (1300,500 125x50), "Reset"
        tap MAIN.Write_Program_Abort.ExecuteCmd
    Label (506,392 46x29), "HOME"
    Label (505,324 42x29), "FOLD"
    Label (487,457 70x29), "APPROACH"
    Label (508,522 46x29), "ORIGIN"
    Button (564,322 58x34)
        OnMouseDown: execute {
            main.Move_Axes.AxisPosition.A1:=-90;
            main.Move_Axes.AxisPosition.A2:=-108;
            main.Move_Axes.AxisPosition.A3:=110;
            main.Move_Axes.AxisPosition.A4:=1;
            main.Move_Axes.AxisPosition.A5:=25;
            main.Move_Axes.AxisPosition.A6:=1;
            gvl_gui.GlobalPositionString := TO_STRING("FOLD");
        }
    Button (564,388 58x34)
        OnMouseClick: execute {
            main.Move_Axes.AxisPosition.A1:=-66;
            main.Move_Axes.AxisPosition.A2:=-90;
            main.Move_Axes.AxisPosition.A3:=70;
            main.Move_Axes.AxisPosition.A4:=1;
            main.Move_Axes.AxisPosition.A5:=15;
            main.Move_Axes.AxisPosition.A6:=1;
            gvl_gui.GlobalPositionString := TO_STRING("Home");
        }
    Button (564,454 58x34)
        OnMouseClick: execute {
            main.Move_Axes.AxisPosition.A1:=1;
            main.Move_Axes.AxisPosition.A2:=-100;
            main.Move_Axes.AxisPosition.A3:=60;
            main.Move_Axes.AxisPosition.A4:=1;
            main.Move_Axes.AxisPosition.A5:=40;
            main.Move_Axes.AxisPosition.A6:=1;
            gvl_gui.GlobalPositionString := TO_STRING("Approach");
        }
    Button (564,520 58x34)
        OnMouseClick: execute {
            main.Move_Axes.AxisPosition.A1:=1;
            main.Move_Axes.AxisPosition.A2:=-70;
            main.Move_Axes.AxisPosition.A3:=50;
            main.Move_Axes.AxisPosition.A4:=1;
            main.Move_Axes.AxisPosition.A5:=20;
            main.Move_Axes.AxisPosition.A6:=1;
            gvl_gui.GlobalPositionString := TO_STRING("Origin");
        }
    Textfield (843,366 121x30), "Go To %s", text variable: GVL_GUI.GlobalPositionString
    Table (543,802 600x43), data array: mxA_Motion.fbKRC_ReadActualPosition.Position
        p3854506369: mxA_Motion.fbKRC_ReadActualPosition.Position.X
        p1892666644: mxA_Motion.fbKRC_ReadActualPosition.Position.Y
        p338671338: mxA_Motion.fbKRC_ReadActualPosition.Position.Z
        p2170511999: mxA_Motion.fbKRC_ReadActualPosition.Position.A
        p3723444502: mxA_Motion.fbKRC_ReadActualPosition.Position.B
        p1218418051: mxA_Motion.fbKRC_ReadActualPosition.Position.C
        p746581629: mxA_Motion.fbKRC_ReadActualPosition.Position.Status
        p3104783080: mxA_Motion.fbKRC_ReadActualPosition.Position.Turn
        p2501879983: mxA_Motion.fbKRC_ReadActualPosition.Position.E1
        p7306298: mxA_Motion.fbKRC_ReadActualPosition.Position.E2
        p1933151965: mxA_Motion.fbKRC_ReadActualPosition.Position.E3
        p3863566920: mxA_Motion.fbKRC_ReadActualPosition.Position.E4
        p2192122294: mxA_Motion.fbKRC_ReadActualPosition.Position.E5
        p400160035: mxA_Motion.fbKRC_ReadActualPosition.Position.E6
        p1757482276: status
        p4088588272: turn
    Table (545,746 599x47), data array: Read_Axes_Velocity.ReadAxesVelocity
        p3854506369: Read_Axes_Velocity.ReadAxesVelocity.AxisGroupIdx
        p1892666644: Read_Axes_Velocity.ReadAxesVelocity.ExecuteCmd
        p338671338: Read_Axes_Velocity.ReadAxesVelocity.Done
        p2170511999: Read_Axes_Velocity.ReadAxesVelocity.Error
        p3723444502: Read_Axes_Velocity.ReadAxesVelocity.ErrorID
        p1218418051: Read_Axes_Velocity.ReadAxesVelocity.A1
        p746581629: Read_Axes_Velocity.ReadAxesVelocity.A2
        p3104783080: Read_Axes_Velocity.ReadAxesVelocity.A3
        p2501879983: Read_Axes_Velocity.ReadAxesVelocity.A4
        p7306298: Read_Axes_Velocity.ReadAxesVelocity.A5
        p1933151965: Read_Axes_Velocity.ReadAxesVelocity.A6
        p3863566920: Read_Axes_Velocity.ReadAxesVelocity.E1
        p2192122294: Read_Axes_Velocity.ReadAxesVelocity.E2
        p400160035: Read_Axes_Velocity.ReadAxesVelocity.E3
        p1265227338: Read_Axes_Velocity.ReadAxesVelocity.E4
        p3726181087: Read_Axes_Velocity.ReadAxesVelocity.E5
        p3136911649: Read_Axes_Velocity.ReadAxesVelocity.E6
        p797552052: Read_Axes_Velocity.ReadAxesVelocity.mxA_ExecuteCommand
    Rectangle (440,751 93x30), "Axes Velocity"
    Lamp1 (977,752 33x33), variable: Read_Axes_Velocity.ReadAxesVelocity.Done, style: Lamp-Lamp1-Green
    Lamp1 (1103,752 33x33), variable: Read_Axes_Velocity.ReadAxesVelocity.Error, style: Lamp-Lamp1-Red
    Rectangle (1007,757 46x22), "DONE"
    Rectangle (1056,757 46x22), "ERROR"
    Rectangle (439,807 93x30), "Tool Position"
END_VISUALIZATION

// ---- VISUs/Motion_Linear.TcVIS
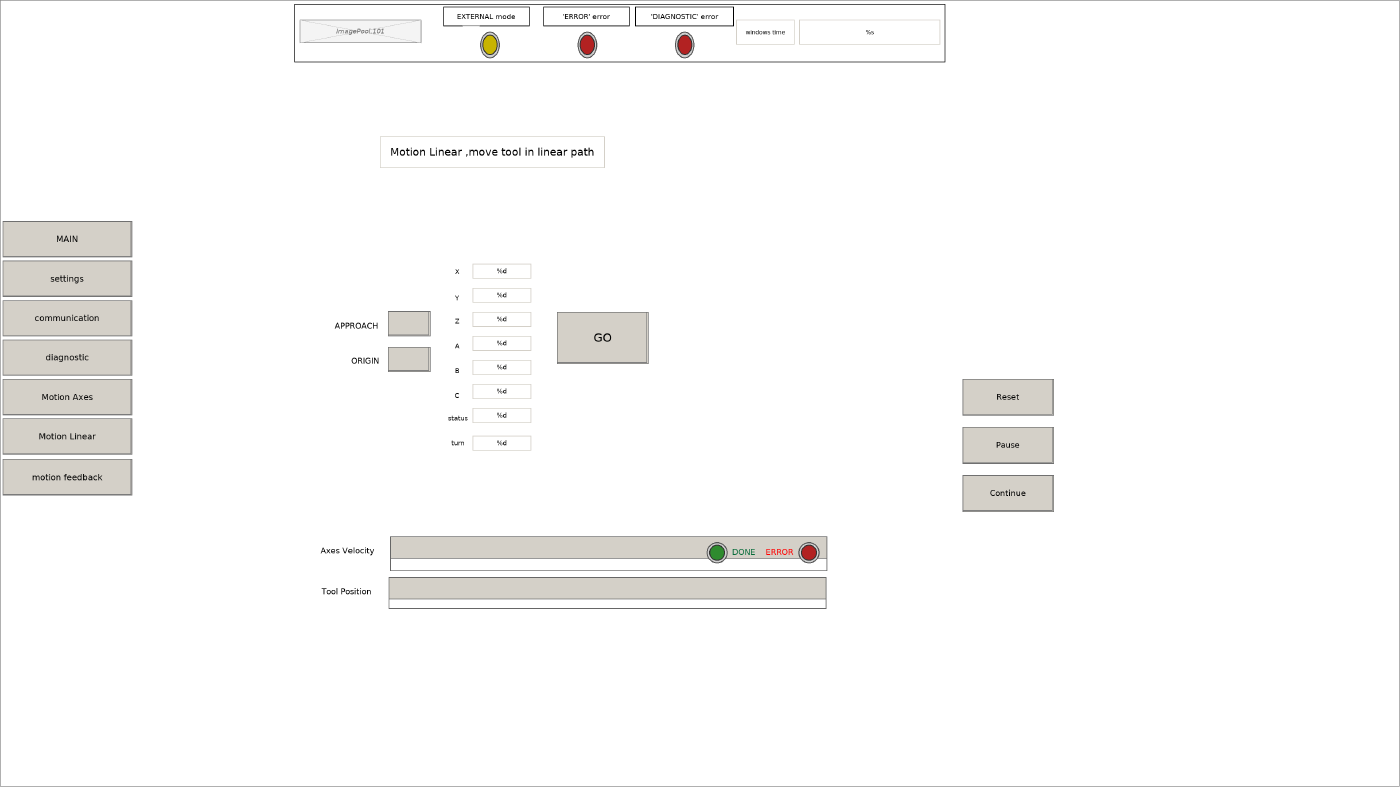
VISUALIZATION Motion_Linear  // 1920x1080
    Frame (400,1 900x90)
        shows MenuTop()
    Frame (0,300 200x400)
        shows MenuMain()
    Textfield (521,187 308x43), "Motion Linear ,move tool in linear path"
    Button (764,428 125x71), "GO"
        tap MAIN.Move_Linear.Execute
    Textfield (648,362 80x20), "%d", text variable: main.LinearTargetPOS.X
    Textfield (648,395 80x20), "%d", text variable: main.LinearTargetPOS.Y
    Textfield (648,428 80x20), "%d", text variable: main.LinearTargetPOS.Z
    Textfield (648,461 80x20), "%d", text variable: main.LinearTargetPOS.A
    Textfield (648,494 80x20), "%d", text variable: main.LinearTargetPOS.B
    Textfield (648,527 80x20), "%d", text variable: main.LinearTargetPOS.C
    Label (610,361 34x24), "X"
    Label (610,397 34x24), "Y"
    Label (610,429 34x24), "Z"
    Label (610,463 34x24), "A"
    Label (610,497 34x24), "B"
    Label (610,531 34x24), "C"
    Label (454,433 70x29), "APPROACH"
    Label (478,481 46x29), "ORIGIN"
    Button (532,427 58x34)
        OnMouseClick: execute {
            //APPROACH COORDINATES:
            main.LinearTargetPOS.X:=974.21;
            main.LinearTargetPOS.y:=-18.91;
            main.LinearTargetPOS.z:=1704.54;
            main.LinearTargetPOS.a:=-97.73;
            main.LinearTargetPOS.b:=88.22;
            main.LinearTargetPOS.c:=-96.10;
            main.LinearTargetPOS.Status :=18;
            main.LinearTargetPOS.Turn:=2;
            //approach
        }
    Button (532,476 58x34)
        OnMouseClick: execute {
            //origin
            main.LinearTargetPOS.X:=1486.29;
            main.LinearTargetPOS.y:=-26.88;
            main.LinearTargetPOS.z:=1422.08;
            main.LinearTargetPOS.a:=-98.31;
            main.LinearTargetPOS.b:=88.04;
            main.LinearTargetPOS.c:=-96.97;
            main.LinearTargetPOS.Status :=18;
            main.LinearTargetPOS.Turn:=2;
        }
    Label (621,326 112x24)
    Textfield (648,560 80x20), "%d", text variable: main.LinearTargetPOS.Status
    Textfield (648,598 80x20), "%d", text variable: main.LinearTargetPOS.Turn
    Label (611,562 34x24), "status"
    Label (611,596 34x24), "turn"
    Button (1320,586 125x50), "Pause"
        tap mxA_Motion.fbAutoDemo.fbKRC_Interrupt.Execute
    Button (1320,652 125x50), "Continue"
        tap mxA_Motion.fbAutoDemo.fbKRC_Continue.Enable
    Button (1320,520 125x50), "Reset"
        tap MAIN.Write_Program_Abort.ExecuteCmd
    Table (533,792 600x43), data array: mxA_Motion.fbKRC_ReadActualPosition.Position
        p3854506369: mxA_Motion.fbKRC_ReadActualPosition.Position.X
        p1892666644: mxA_Motion.fbKRC_ReadActualPosition.Position.Y
        p338671338: mxA_Motion.fbKRC_ReadActualPosition.Position.Z
        p2170511999: mxA_Motion.fbKRC_ReadActualPosition.Position.A
        p3723444502: mxA_Motion.fbKRC_ReadActualPosition.Position.B
        p1218418051: mxA_Motion.fbKRC_ReadActualPosition.Position.C
        p746581629: mxA_Motion.fbKRC_ReadActualPosition.Position.Status
        p3104783080: mxA_Motion.fbKRC_ReadActualPosition.Position.Turn
        p2501879983: mxA_Motion.fbKRC_ReadActualPosition.Position.E1
        p7306298: mxA_Motion.fbKRC_ReadActualPosition.Position.E2
        p1933151965: mxA_Motion.fbKRC_ReadActualPosition.Position.E3
        p3863566920: mxA_Motion.fbKRC_ReadActualPosition.Position.E4
        p2192122294: mxA_Motion.fbKRC_ReadActualPosition.Position.E5
        p400160035: mxA_Motion.fbKRC_ReadActualPosition.Position.E6
        p1757482276: status
        p4088588272: turn
    Table (535,736 599x47), data array: Read_Axes_Velocity.ReadAxesVelocity
        p3854506369: Read_Axes_Velocity.ReadAxesVelocity.AxisGroupIdx
        p1892666644: Read_Axes_Velocity.ReadAxesVelocity.ExecuteCmd
        p338671338: Read_Axes_Velocity.ReadAxesVelocity.Done
        p2170511999: Read_Axes_Velocity.ReadAxesVelocity.Error
        p3723444502: Read_Axes_Velocity.ReadAxesVelocity.ErrorID
        p1218418051: Read_Axes_Velocity.ReadAxesVelocity.A1
        p746581629: Read_Axes_Velocity.ReadAxesVelocity.A2
        p3104783080: Read_Axes_Velocity.ReadAxesVelocity.A3
        p2501879983: Read_Axes_Velocity.ReadAxesVelocity.A4
        p7306298: Read_Axes_Velocity.ReadAxesVelocity.A5
        p1933151965: Read_Axes_Velocity.ReadAxesVelocity.A6
        p3863566920: Read_Axes_Velocity.ReadAxesVelocity.E1
        p2192122294: Read_Axes_Velocity.ReadAxesVelocity.E2
        p400160035: Read_Axes_Velocity.ReadAxesVelocity.E3
        p1265227338: Read_Axes_Velocity.ReadAxesVelocity.E4
        p3726181087: Read_Axes_Velocity.ReadAxesVelocity.E5
        p3136911649: Read_Axes_Velocity.ReadAxesVelocity.E6
        p797552052: Read_Axes_Velocity.ReadAxesVelocity.mxA_ExecuteCommand
    Rectangle (430,741 93x30), "Axes Velocity"
    Lamp1 (967,742 33x33), variable: Read_Axes_Velocity.ReadAxesVelocity.Done, style: Lamp-Lamp1-Green
    Lamp1 (1093,742 33x33), variable: Read_Axes_Velocity.ReadAxesVelocity.Error, style: Lamp-Lamp1-Red
    Rectangle (997,747 46x22), "DONE"
    Rectangle (1046,747 46x22), "ERROR"
    Rectangle (429,797 93x30), "Tool Position"
END_VISUALIZATION

// ---- VISUs/Motion_FBK.TcVIS
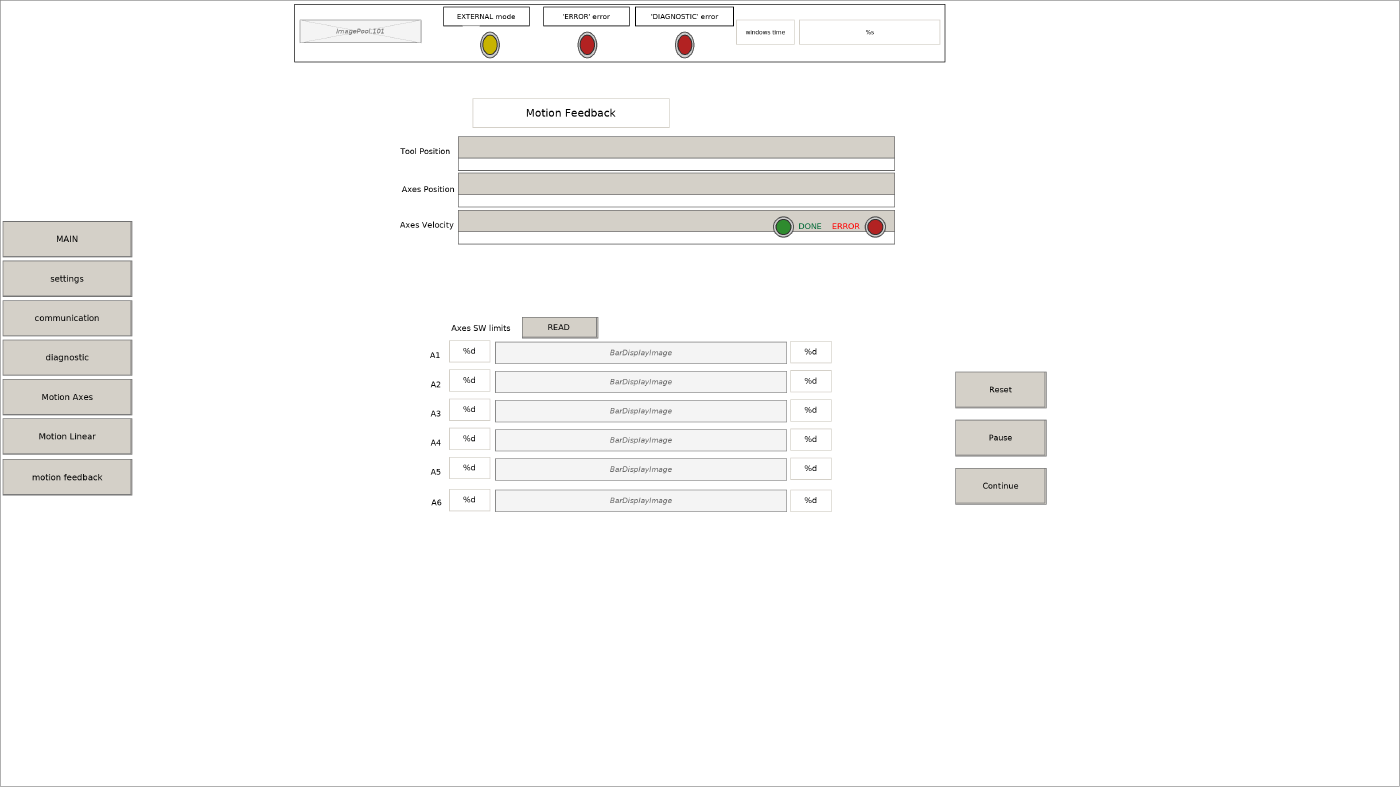
VISUALIZATION Motion_FBK  // 1920x1080
    Frame (400,1 900x90)
        shows MenuTop()
    Frame (0,300 200x400)
        shows MenuMain()
    Textfield (648,135 270x40), "Motion Feedback"
    Table (628,237 599x47), data array: GVL.HMI_ActualAxisPosition
        p3854506369: GVL.HMI_ActualAxisPosition.A1
        p1892666644: GVL.HMI_ActualAxisPosition.A2
        p338671338: GVL.HMI_ActualAxisPosition.A3
        p2170511999: GVL.HMI_ActualAxisPosition.A4
        p3723444502: GVL.HMI_ActualAxisPosition.A5
        p1218418051: GVL.HMI_ActualAxisPosition.A6
        p746581629: GVL.HMI_ActualAxisPosition.E1
        p3104783080: GVL.HMI_ActualAxisPosition.E2
        p2501879983: GVL.HMI_ActualAxisPosition.E3
        p7306298: GVL.HMI_ActualAxisPosition.E4
        p1933151965: GVL.HMI_ActualAxisPosition.E5
        p3863566920: GVL.HMI_ActualAxisPosition.E6
        p2192122294: ActualKarthPositon.E5
        p400160035: ActualKarthPositon.E6
    Table (628,187 599x47), data array: mxA_Motion.fbKRC_ReadActualPosition.Position
        p3854506369: mxA_Motion.fbKRC_ReadActualPosition.Position.X
        p1892666644: mxA_Motion.fbKRC_ReadActualPosition.Position.Y
        p338671338: mxA_Motion.fbKRC_ReadActualPosition.Position.Z
        p2170511999: mxA_Motion.fbKRC_ReadActualPosition.Position.A
        p3723444502: mxA_Motion.fbKRC_ReadActualPosition.Position.B
        p1218418051: mxA_Motion.fbKRC_ReadActualPosition.Position.C
        p746581629: mxA_Motion.fbKRC_ReadActualPosition.Position.Status
        p3104783080: mxA_Motion.fbKRC_ReadActualPosition.Position.Turn
        p2501879983: mxA_Motion.fbKRC_ReadActualPosition.Position.E1
        p7306298: mxA_Motion.fbKRC_ReadActualPosition.Position.E2
        p1933151965: mxA_Motion.fbKRC_ReadActualPosition.Position.E3
        p3863566920: mxA_Motion.fbKRC_ReadActualPosition.Position.E4
        p2192122294: mxA_Motion.fbKRC_ReadActualPosition.Position.E5
        p400160035: mxA_Motion.fbKRC_ReadActualPosition.Position.E6
        p4092479075: Rx
        p2237128397: Ry
        p505689113: Rz
        p1757482276: status
        p4088588272: turn
    Rectangle (537,193 93x30), "Tool Position"
    Rectangle (541,245 93x30), "Axes Position"
    BarDisplayImage (679,469 400x30), value: mxA_Motion.fbKRC_ReadActualAxisPosition.A1, style: BarDisplayImage-Gray, scale format: %.1f, scale -180..180
    BarDisplayImage (679,509 400x30), value: mxA_Motion.fbKRC_ReadActualAxisPosition.A2, style: BarDisplayImage-Gray, scale format: %.1f, scale -180..180
    BarDisplayImage (679,549 400x30), value: mxA_Motion.fbKRC_ReadActualAxisPosition.A3, style: BarDisplayImage-Gray, scale format: %.1f, scale -180..180
    BarDisplayImage (679,589 400x30), value: mxA_Motion.fbKRC_ReadActualAxisPosition.A4, style: BarDisplayImage-Gray, scale format: %.1f, scale -360..360
    BarDisplayImage (679,629 400x30), value: mxA_Motion.fbKRC_ReadActualAxisPosition.A5, style: BarDisplayImage-Gray, scale format: %.1f, scale -180..180
    BarDisplayImage (679,672 400x30), value: mxA_Motion.fbKRC_ReadActualAxisPosition.A6, style: BarDisplayImage-Gray, scale format: %.1f, scale -360..360
    Label (580,476 34x24), "A1"
    Label (581,516 34x24), "A2"
    Label (581,556 34x24), "A3"
    Label (581,596 34x24), "A4"
    Label (581,636 34x24), "A5"
    Label (582,678 34x24), "A6"
    Rectangle (603,430 113x41), "Axes SW limits"
    Textfield (1084,468 56x30), "%d", text variable: MAIN.Read_Axes_SW_Limts.A1_Max
    Textfield (1084,508 56x30), "%d", text variable: MAIN.Read_Axes_SW_Limts.A2_Max
    Textfield (1084,548 56x30), "%d", text variable: MAIN.Read_Axes_SW_Limts.A3_Max
    Textfield (1084,588 56x30), "%d", text variable: MAIN.Read_Axes_SW_Limts.A4_Max
    Textfield (1084,628 56x30), "%d", text variable: MAIN.Read_Axes_SW_Limts.A5_Max
    Textfield (1084,672 56x30), "%d", text variable: MAIN.Read_Axes_SW_Limts.A6_Max
    Textfield (616,467 56x30), "%d", text variable: MAIN.Read_Axes_SW_Limts.A1_Min
    Textfield (616,507 56x30), "%d", text variable: MAIN.Read_Axes_SW_Limts.A2_Min
    Textfield (616,547 56x30), "%d", text variable: MAIN.Read_Axes_SW_Limts.A3_Min
    Textfield (616,587 56x30), "%d", text variable: MAIN.Read_Axes_SW_Limts.A4_Min
    Textfield (616,627 56x30), "%d", text variable: MAIN.Read_Axes_SW_Limts.A5_Min
    Textfield (616,671 56x30), "%d", text variable: MAIN.Read_Axes_SW_Limts.A6_Min
    Button (716,435 104x29), "READ"
        OnMouseClick: toggle MAIN.Read_Axes_SW_Limts.ExecuteCmd
    Button (1310,576 125x50), "Pause"
        tap mxA_Motion.fbAutoDemo.fbKRC_Interrupt.Execute
    Button (1310,642 125x50), "Continue"
        tap mxA_Motion.fbAutoDemo.fbKRC_Continue.Enable
    Button (1310,510 125x50), "Reset"
        tap MAIN.Write_Program_Abort.ExecuteCmd
    Table (628,288 599x47), data array: Read_Axes_Velocity.ReadAxesVelocity
        p3854506369: Read_Axes_Velocity.ReadAxesVelocity.AxisGroupIdx
        p1892666644: Read_Axes_Velocity.ReadAxesVelocity.ExecuteCmd
        p338671338: Read_Axes_Velocity.ReadAxesVelocity.Done
        p2170511999: Read_Axes_Velocity.ReadAxesVelocity.Error
        p3723444502: Read_Axes_Velocity.ReadAxesVelocity.ErrorID
        p1218418051: Read_Axes_Velocity.ReadAxesVelocity.A1
        p746581629: Read_Axes_Velocity.ReadAxesVelocity.A2
        p3104783080: Read_Axes_Velocity.ReadAxesVelocity.A3
        p2501879983: Read_Axes_Velocity.ReadAxesVelocity.A4
        p7306298: Read_Axes_Velocity.ReadAxesVelocity.A5
        p1933151965: Read_Axes_Velocity.ReadAxesVelocity.A6
        p3863566920: Read_Axes_Velocity.ReadAxesVelocity.E1
        p2192122294: Read_Axes_Velocity.ReadAxesVelocity.E2
        p400160035: Read_Axes_Velocity.ReadAxesVelocity.E3
        p1265227338: Read_Axes_Velocity.ReadAxesVelocity.E4
        p3726181087: Read_Axes_Velocity.ReadAxesVelocity.E5
        p3136911649: Read_Axes_Velocity.ReadAxesVelocity.E6
        p797552052: Read_Axes_Velocity.ReadAxesVelocity.mxA_ExecuteCommand
    Rectangle (539,294 93x30), "Axes Velocity"
    Lamp1 (1058,295 33x33), variable: Read_Axes_Velocity.ReadAxesVelocity.Done, style: Lamp-Lamp1-Green
    Lamp1 (1184,295 33x33), variable: Read_Axes_Velocity.ReadAxesVelocity.Error, style: Lamp-Lamp1-Red
    Rectangle (1088,300 46x22), "DONE"
    Rectangle (1137,300 46x22), "ERROR"
END_VISUALIZATION

// ---- VISUs/MenuMain.TcVIS
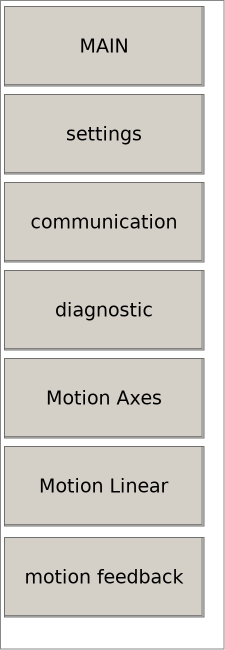
VISUALIZATION MenuMain  // 225x650
    Button (4,94 200x80), "settings"
        OnMouseClick: change screen: APP_Settings
    Button (4,182 200x80), "communication"
        OnMouseClick: change screen: communication
    Button (4,358 200x80), "Motion Axes"
        OnMouseClick: change screen: Motion_Axes
    Button (4,537 200x80), "motion feedback"
        OnMouseClick: change screen: Motion_FBK
    Button (4,6 200x80), "MAIN"
        OnMouseClick: change screen: MainScreen
    Button (4,446 200x80), "Motion Linear"
        OnMouseClick: change screen: Motion_Linear
    Button (4,270 200x80), "diagnostic"
        OnMouseClick: change screen: diagnostic
END_VISUALIZATION

// ---- VISUs/MenuTop.TcVIS
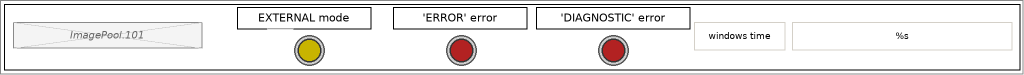
VISUALIZATION MenuTop  // 1024x75
    RoundedRectangle (4,4 1016x66)
    Lamp1 (292,33 35x35), variable: MAIN.fbKRC_AutomaticExternal.IO_ACTCONF, style: Lamp-Lamp1-Yellow
    Lamp1 (444,33 35x35), variable: MAIN.fbKRC_Error.Error, style: Lamp-Lamp1-Red
    Textfield (792,22 220x28), "%s", text variable: GVL_PLC.String_WindowsTime
    Textfield (694,22 91x28), "windows time"
    Lamp1 (596,33 35x35), variable: MAIN.fbKRC_Diag.Error, style: Lamp-Lamp1-Red
    RoundedRectangle (237,7 134x22), "EXTERNAL mode"
    RoundedRectangle (393,7 134x22), "'ERROR' error"
    RoundedRectangle (536,7 154x22), "'DIAGNOSTIC' error"
    Image (13,22 189x26), image: ImagePool.101
    Image (267,28 26x1)
END_VISUALIZATION

// ---- VISUs/HMI_dmeo.TcVIS
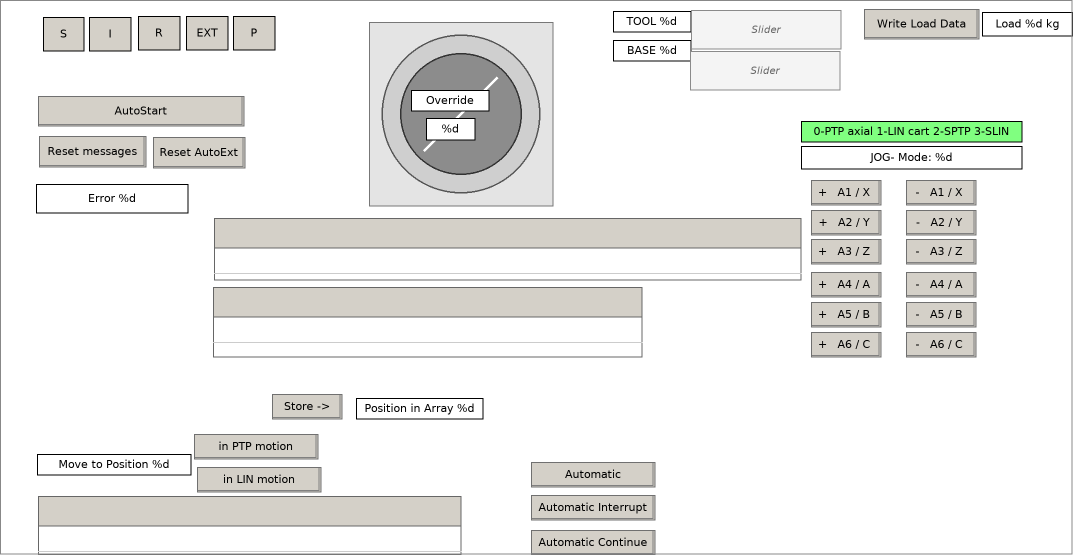
VISUALIZATION HMI_dmeo  // 1073x555
    Potentiometer360 (362,22 198x184), variable: GVL.nOverrideGlobal, style: Potentiometer-Potentiometer360-Gray, scale format: %d, scale 0..100
    Rectangle (411,90 78x21), "Override"
    Rectangle (426,118 49x22), "%d", text variable: GVL.nOverrideGlobal
        OnMouseClick: write the text variable via VisuDialogs.Numpad
    Button (38,96 206x30), "AutoStart", colour toggle: MAIN.bAutostartDone
        tap GVL.HMI_AutoStart
    Button (39,136 107x31), "Reset messages"
        tap GVL.HMI_MessageReset
    Rectangle (613,11 78x21), "TOOL %d", text variable: GVL.HMI_TOOL
        OnMouseClick: write the text variable via Default, min 1, max 16
    Rectangle (613,40 78x21), "BASE %d", text variable: GVL.HMI_BASE
        OnMouseClick: write the text variable via Default, min 1, max 16
    Slider (691,10 150x39), variable: GVL.HMI_TOOL, scale 0..5
    Slider (690,51 150x39), variable: GVL.HMI_BASE, scale 0..5
    Line (808,124)
    Rectangle (801,146 221x23), "JOG- Mode: %d", text variable: mxA_Motion.nJogMoveType
        OnMouseClick: write the text variable via Default, min 0, max 3
    Button (811,180 70x25), "+ A1 / X"
        tap mxA_Motion.bJogA1_P
    Button (906,180 70x25), "- A1 / X"
        tap mxA_Motion.bJogA1_M
    Button (864,9 115x30), "Write Load Data"
        tap GVL.HMI_WriteLoadData
    Rectangle (982,12 91x24), "Load %d kg", text variable: GVL.HMI_LOAD
        OnMouseClick: write the text variable via Default
    Rectangle (801,121 221x21), "0-PTP axial 1-LIN cart 2-SPTP 3-SLIN"
    Button (811,210 70x25), "+ A2 / Y"
        tap mxA_Motion.bJogA2_P
    Button (906,210 70x25), "- A2 / Y"
        tap mxA_Motion.bJogA2_M
    Button (811,239 70x25), "+ A3 / Z"
        tap mxA_Motion.bJogA3_P
    Button (906,239 70x25), "- A3 / Z"
        tap mxA_Motion.bJogA3_M
    Button (811,272 70x25), "+ A4 / A"
        tap mxA_Motion.bJogA4_P
    Button (906,272 70x25), "- A4 / A"
        tap mxA_Motion.bJogA4_M
    Button (811,302 70x25), "+ A5 / B"
        tap mxA_Motion.bJogA5_P
    Button (906,302 70x25), "- A5 / B"
        tap mxA_Motion.bJogA5_M
    Button (811,332 70x25), "+ A6 / C"
        tap mxA_Motion.bJogA6_P
    Button (906,332 70x25), "- A6 / C"
        tap mxA_Motion.bJogA6_M
    Rectangle (43,17 41x34), "S", colour toggle: GVL.HMI_Error_SINT
    Rectangle (233,16 42x34), "P", colour toggle: GVL.HMI_Error_ProConOS
    Rectangle (89,17 42x34), "I", colour toggle: GVL.HMI_DrivesNotReady
    Rectangle (138,16 42x34), "R", colour toggle: MAIN.bAutostartDispActive
    Rectangle (186,16 42x34), "EXT", colour toggle: GVL.HMI_AutoEXT
    Rectangle (36,184 152x29), "Error %d", text variable: GVL.HMI_Error_General_ID, colour toggle: GVL.HMI_Error_General
    Table (214,218 587x62), data array: GVL.HMI_ActualCartPos
        p3854506369: GVL.HMI_ActualCartPos.X
        p1892666644: GVL.HMI_ActualCartPos.Y
        p338671338: GVL.HMI_ActualCartPos.Z
        p2170511999: GVL.HMI_ActualCartPos.A
        p3723444502: GVL.HMI_ActualCartPos.B
        p1218418051: GVL.HMI_ActualCartPos.C
        p746581629: GVL.HMI_ActualCartPos.Status
        p3104783080: GVL.HMI_ActualCartPos.Turn
        p2501879983: GVL.HMI_ActualCartPos.E1
        p7306298: GVL.HMI_ActualCartPos.E2
        p1933151965: GVL.HMI_ActualCartPos.E3
        p3863566920: GVL.HMI_ActualCartPos.E4
        p2192122294: GVL.HMI_ActualCartPos.E5
        p400160035: GVL.HMI_ActualCartPos.E6
    Table (213,287 429x70), data array: GVL.HMI_ActualAxisPosition
        p3854506369: GVL.HMI_ActualAxisPosition.A1
        p1892666644: GVL.HMI_ActualAxisPosition.A2
        p338671338: GVL.HMI_ActualAxisPosition.A3
        p2170511999: GVL.HMI_ActualAxisPosition.A4
        p3723444502: GVL.HMI_ActualAxisPosition.A5
        p1218418051: GVL.HMI_ActualAxisPosition.A6
        p746581629: GVL.HMI_ActualAxisPosition.E1
        p3104783080: GVL.HMI_ActualAxisPosition.E2
        p2501879983: GVL.HMI_ActualAxisPosition.E3
        p7306298: GVL.HMI_ActualAxisPosition.E4
        p1933151965: GVL.HMI_ActualAxisPosition.E5
        p3863566920: GVL.HMI_ActualAxisPosition.E6
        p2192122294: ActualKarthPositon.E5
        p400160035: ActualKarthPositon.E6
    Button (153,137 92x31), "Reset AutoExt"
        tap MAIN.bAutoExternReset
    Rectangle (356,398 127x21), "Position in Array %d", text variable: GVL.HMI_TouchUpIndex
        OnMouseClick: write the text variable via Default, min 1, max 100
    Button (272,394 70x25), "Store ->"
        tap GVL.HMI_TouchUpStoreNow
    Rectangle (37,454 154x21), "Move to Position %d", text variable: mxA_Motion.nMove_PositonMode_Pos
        OnMouseClick: write the text variable via Default, min 1, max 16
    Button (197,467 124x25), "in LIN motion"
        tap mxA_Motion.bMoveLinar_PositonMode
    Table (38,496 423x59), data array: GVL.aPosArray[mxA_Motion.nMove_PositonMode_Pos].E6AXIS
        p2192122294: ActualKarthPositon.E5
        p400160035: ActualKarthPositon.E6
        p3854506369: GVL.aPosArray[mxA_Motion.nMove_PositonMode_Pos].E6AXIS.A1
        p1892666644: GVL.aPosArray[mxA_Motion.nMove_PositonMode_Pos].E6AXIS.A2
        p338671338: GVL.aPosArray[mxA_Motion.nMove_PositonMode_Pos].E6AXIS.A3
        p2170511999: GVL.aPosArray[mxA_Motion.nMove_PositonMode_Pos].E6AXIS.A4
        p3723444502: GVL.aPosArray[mxA_Motion.nMove_PositonMode_Pos].E6AXIS.A5
        p1218418051: GVL.aPosArray[mxA_Motion.nMove_PositonMode_Pos].E6AXIS.A6
        p746581629: GVL.aPosArray[mxA_Motion.nMove_PositonMode_Pos].E6AXIS.E1
        p3104783080: GVL.aPosArray[mxA_Motion.nMove_PositonMode_Pos].E6AXIS.E2
        p2501879983: GVL.aPosArray[mxA_Motion.nMove_PositonMode_Pos].E6AXIS.E3
        p7306298: GVL.aPosArray[mxA_Motion.nMove_PositonMode_Pos].E6AXIS.E4
        p1933151965: GVL.aPosArray[mxA_Motion.nMove_PositonMode_Pos].E6AXIS.E5
        p3863566920: GVL.aPosArray[mxA_Motion.nMove_PositonMode_Pos].E6AXIS.E6
    Button (194,434 124x25), "in PTP motion"
        tap mxA_Motion.bMovePTP_PositonMode
    Button (531,462 124x25), "Automatic", colour toggle: mxA_Motion.bExecAutoDemo
        toggle mxA_Motion.bExecAutoDemo
    Button (531,495 124x25), "Automatic Interrupt"
        tap mxA_Motion.fbAutoDemo.fbKRC_Interrupt.Execute
    Button (531,530 124x25), "Automatic Continue"
        tap mxA_Motion.fbAutoDemo.fbKRC_Continue.Enable
END_VISUALIZATION

// ---- VISUs/MainScreen.TcVIS
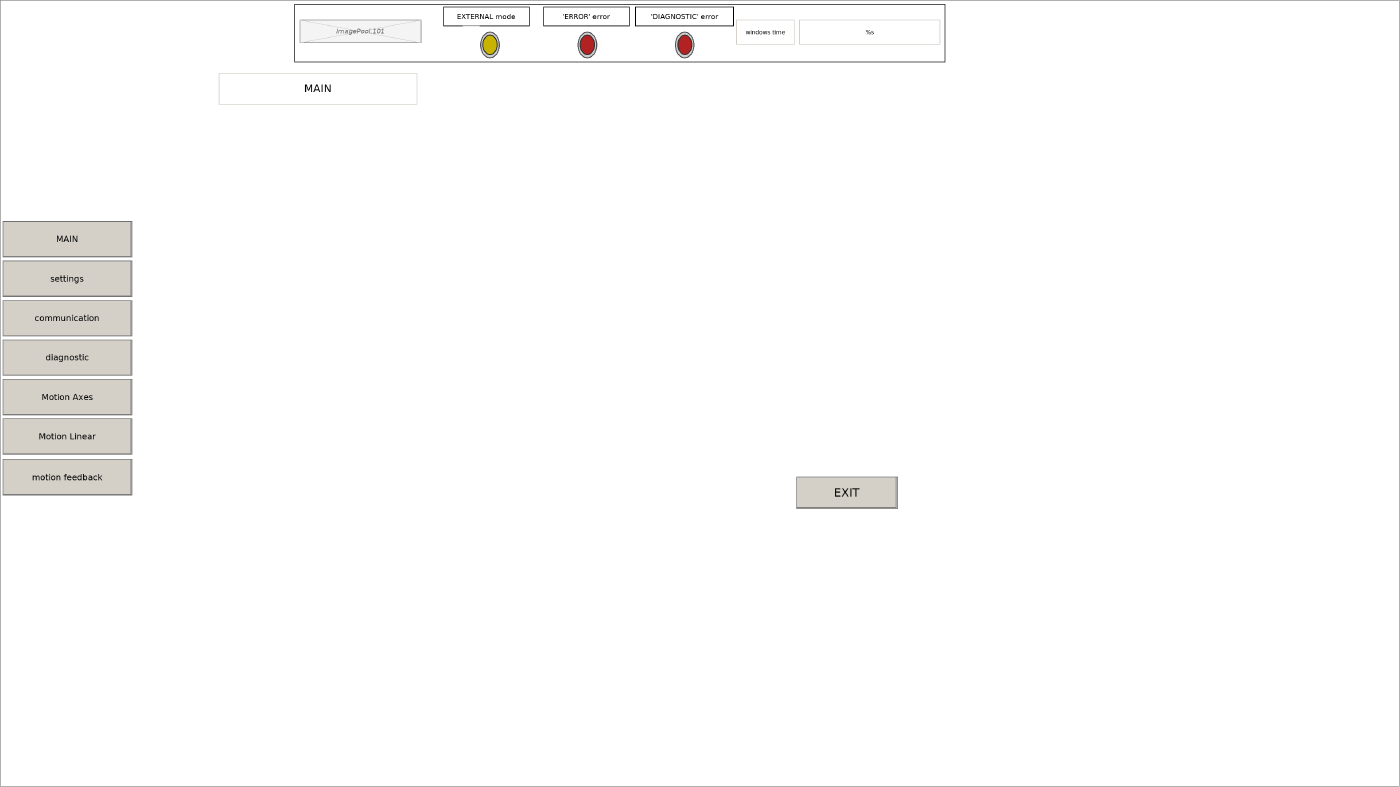
VISUALIZATION MainScreen  // 1920x1080
    Frame (400,1 900x90)
        shows MenuTop()
    Frame (0,300 200x400)
        shows MenuMain()
    Textfield (300,100 272x43), "MAIN"
    Button (1092,654 139x44), "EXIT"
        OnMouseClick: ExecuteCommand ExecuteCommand=ExecuteCommand=[Command=ExecuteClientProgram, Value='TASKKILL /F /IM', Value2='Tc3PlcHmi.exe']
END_VISUALIZATION

// ---- VISUs/Text Lists/CoorSys.TcTLO
TEXTLIST CoorSys
  1 = 'robot'
  2 = 'couch'
  3 = 'calibration'
  4 = 'spare'
  5 = 'default'
   = ''
END_TEXTLIST

// ---- VISUs/Text Lists/GlobalPositions.TcTLO
TEXTLIST GlobalPositions
  1 = 'Fold'
  2 = 'Home'
  3 = 'Approach'
  4 = 'Origin'
   = ''
END_TEXTLIST

// ---- VISUs/Text Lists/ToolNumber.TcTLO
TEXTLIST ToolNumber
  1 = 'laser'
  2 = 'screw'
  3 = 'demo'
  4 = 'lens'
  5 = 'spare'
   = ''
END_TEXTLIST
